  MoveL 604 to (474.95, 542.05, 8) mm, rotated rx 180 ry 0 rz 160 deg; joints [12.107, 76.051, -6.666, -146.162, 72.648, 168.694]
  Set speed (17.5 mm/s)
  Call Extruder(1520.11430)
  MoveL 605 to (474.5, 541.77, 8) mm, rotated rx 180 ry 0 rz 160 deg; joints [12.084, 75.99, -6.51, -146.202, 72.722, 168.756]
  Set speed (17.5 mm/s)
  Call Extruder(1525.02025)
  MoveL 606 to (473.22, 540.96, 8) mm, rotated rx 180 ry 0 rz 160 deg; joints [12.014, 75.813, -6.063, -146.32, 72.934, 168.934]
  Set speed (17.5 mm/s)
  Call Extruder(1527.82496)
  MoveL 607 to (472.5, 540.48, 8) mm, rotated rx 180 ry 0 rz 160 deg; joints [11.972, 75.714, -5.811, -146.39, 73.053, 169.035]
  Set speed (17.4 mm/s)
  Call Extruder(1533.06308)
  MoveL 608 to (471.18, 539.55, 8) mm, rotated rx -180 ry 0 rz 160 deg; joints [11.887, 75.532, -5.348, -146.524, 73.271, 169.223]
  Set speed (17.4 mm/s)
  Call Extruder(1536.34508)
  MoveL 609 to (470.36, 538.94, 8) mm, rotated rx 180 ry 0 rz 160 deg; joints [11.83, 75.421, -5.064, -146.611, 73.405, 169.339]
  Set speed (17.4 mm/s)
  Call Extruder(1538.57380)
  MoveL 610 to (469.82, 538.52, 8) mm, rotated rx 180 ry 0 rz 160 deg; joints [11.79, 75.346, -4.872, -146.671, 73.495, 169.418]
  Set speed (17.5 mm/s)
  Call Extruder(1541.82142)
  MoveL 611 to (469.03, 537.89, 8) mm, rotated rx -180 ry 0 rz 160 deg; joints [11.729, 75.239, -4.597, -146.761, 73.625, 169.532]
  Set speed (17.5 mm/s)
  Call Extruder(1547.90773)
  MoveL 612 to (467.59, 536.68, 8) mm, rotated rx 180 ry 0 rz 160 deg; joints [11.608, 75.042, -4.09, -146.934, 73.863, 169.743]
  Set speed (17.5 mm/s)
  Call Extruder(1552.51952)
  MoveL 613 to (466.54, 535.71, 8) mm, rotated rx 180 ry 0 rz 160 deg; joints [11.509, 74.899, -3.717, -147.071, 74.037, 169.901]
  Set speed (17.4 mm/s)
  Call Extruder(1558.05894)
  MoveL 614 to (465.31, 534.52, 8) mm, rotated rx -180 ry 0 rz 160 deg; joints [11.384, 74.731, -3.281, -147.241, 74.241, 170.087]
  Set speed (17.5 mm/s)
  Call Extruder(1561.63478)
  MoveL 615 to (464.54, 533.73, 8) mm, rotated rx 180 ry 0 rz 160 deg; joints [11.299, 74.625, -3.007, -147.353, 74.369, 170.206]
  Call Extruder(1565.31804)
  MoveL 616 to (463.76, 532.89, 8) mm, rotated rx -180 ry 0 rz 160 deg; joints [11.208, 74.519, -2.73, -147.472, 74.497, 170.326]
  Set speed (17.5 mm/s)
  Call Extruder(1568.71161)
  MoveL 617 to (463.07, 532.11, 8) mm, rotated rx 180 ry 0 rz 160 deg; joints [11.122, 74.424, -2.479, -147.583, 74.614, 170.436]
  Call Extruder(0.00000)
  Set speed (17.4 mm/s)
  Call Extruder(3.82302)
  MoveL 618 to (462.3, 531.2, 8) mm, rotated rx 180 ry 0 rz 160 deg; joints [11.021, 74.319, -2.204, -147.711, 74.741, 170.558]
  Set speed (17.5 mm/s)
  Call Extruder(8.69578)
  MoveL 619 to (461.36, 530.03, 8) mm, rotated rx 180 ry 0 rz 160 deg; joints [10.888, 74.19, -1.863, -147.878, 74.898, 170.71]
  Set speed (17.5 mm/s)
  Call Extruder(11.81632)
  MoveL 620 to (460.77, 529.26, 8) mm, rotated rx 180 ry 0 rz 160 deg; joints [10.799, 74.109, -1.65, -147.988, 74.996, 170.807]
  Set speed (17.5 mm/s)
  Call Extruder(16.00361)
  MoveL 621 to (460.01, 528.21, 8) mm, rotated rx 180 ry 0 rz 160 deg; joints [10.677, 74.004, -1.372, -148.137, 75.124, 170.934]
  Set speed (17.5 mm/s)
  Call Extruder(19.39363)
  MoveL 622 to (459.42, 527.35, 8) mm, rotated rx 180 ry 0 rz 160 deg; joints [10.575, 73.922, -1.153, -148.26, 75.224, 171.035]
  Set speed (17.5 mm/s)
  Call Extruder(23.27967)
  MoveL 623 to (458.76, 526.34, 8) mm, rotated rx 180 ry 0 rz 160 deg; joints [10.456, 73.83, -0.91, -148.403, 75.335, 171.148]
  Set speed (17.5 mm/s)
  Call Extruder(28.16959)
  MoveL 624 to (457.96, 525.05, 8) mm, rotated rx 180 ry 0 rz 160 deg; joints [10.3, 73.72, -0.614, -148.587, 75.469, 171.288]
  Call Extruder(32.04491)
  MoveL 625 to (457.36, 524.02, 8) mm, rotated rx -180 ry 0 rz 160 deg; joints [10.174, 73.635, -0.388, -148.735, 75.571, 171.397]
  Set speed (17.5 mm/s)
  Call Extruder(35.64970)
  MoveL 626 to (456.83, 523.04, 8) mm, rotated rx 180 ry 0 rz 160 deg; joints [10.053, 73.559, -0.184, -148.875, 75.662, 171.495]
  Call Extruder(38.75076)
  MoveL 627 to (456.38, 522.19, 8) mm, rotated rx -180 ry 0 rz 160 deg; joints [9.948, 73.497, -0.015, -148.997, 75.738, 171.579]
  Set speed (17.4 mm/s)
  Call Extruder(42.04623)
  MoveL 628 to (455.93, 521.28, 8) mm, rotated rx 180 ry 0 rz 160 deg; joints [9.833, 73.432, 0.159, -149.128, 75.815, 171.665]
  Set speed (17.4 mm/s)
  Call Extruder(45.26649)
  MoveL 629 to (455.51, 520.38, 8) mm, rotated rx 180 ry 0 rz 160 deg; joints [9.719, 73.371, 0.323, -149.258, 75.887, 171.748]
  Set speed (17.4 mm/s)
  Call Extruder(48.51642)
  MoveL 630 to (455.1, 519.46, 8) mm, rotated rx 180 ry 0 rz 160 deg; joints [9.603, 73.312, 0.484, -149.389, 75.958, 171.831]
  Set speed (17.4 mm/s)
  Call Extruder(52.84820)
  MoveL 631 to (454.58, 518.22, 8) mm, rotated rx -180 ry 0 rz 160 deg; joints [9.444, 73.236, 0.689, -149.568, 76.047, 171.937]
  Set speed (17.5 mm/s)
  Call Extruder(59.01689)
  MoveL 632 to (453.9, 516.44, 8) mm, rotated rx -180 ry 0 rz 160 deg; joints [9.213, 73.135, 0.964, -149.825, 76.164, 172.084]
  Set speed (17.5 mm/s)
  Call Extruder(61.45313)
  MoveL 633 to (453.66, 515.72, 8) mm, rotated rx -180 ry 0 rz 160 deg; joints [9.119, 73.098, 1.064, -149.928, 76.207, 172.14]
  Set speed (17.4 mm/s)
  Call Extruder(67.12764)
  MoveL 634 to (453.12, 514.05, 8) mm, rotated rx 180 ry 0 rz 160 deg; joints [8.899, 73.015, 1.29, -150.17, 76.301, 172.267]
  Set speed (17.4 mm/s)
  Call Extruder(71.17621)
  MoveL 635 to (452.78, 512.85, 8) mm, rotated rx -180 ry 0 rz 160 deg; joints [8.739, 72.961, 1.438, -150.345, 76.361, 172.353]
  Set speed (17.4 mm/s)
  Call Extruder(74.29378)
  MoveL 636 to (452.53, 511.92, 8) mm, rotated rx -180 ry 0 rz 160 deg; joints [8.615, 72.921, 1.548, -150.48, 76.405, 172.419]
  Set speed (17.4 mm/s)
  Call Extruder(77.03216)
  MoveL 637 to (452.34, 511.1, 8) mm, rotated rx 180 ry 0 rz 160 deg; joints [8.504, 72.888, 1.637, -150.6, 76.44, 172.474]
  Set speed (17.4 mm/s)
  Call Extruder(81.46566)
  MoveL 638 to (452.05, 509.76, 8) mm, rotated rx 180 ry 0 rz 160 deg; joints [8.324, 72.838, 1.775, -150.794, 76.493, 172.561]
  Set speed (17.4 mm/s)
  Call Extruder(87.40179)
  MoveL 639 to (451.72, 507.96, 8) mm, rotated rx 180 ry 0 rz 160 deg; joints [8.078, 72.778, 1.94, -151.057, 76.553, 172.672]
  Set speed (17.5 mm/s)
  Call Extruder(91.56460)
  MoveL 640 to (451.53, 506.68, 8) mm, rotated rx -180 ry 0 rz 160 deg; joints [7.903, 72.741, 2.043, -151.243, 76.589, 172.746]
  Set speed (17.5 mm/s)
  Call Extruder(93.86761)
  MoveL 641 to (451.43, 505.98, 8) mm, rotated rx 180 ry 0 rz 160 deg; joints [7.806, 72.721, 2.097, -151.346, 76.606, 172.786]
  Set speed (17.4 mm/s)
  Call Extruder(100.33911)
  MoveL 642 to (451.23, 503.99, 8) mm, rotated rx -180 ry 0 rz 160 deg; joints [7.53, 72.673, 2.229, -151.636, 76.646, 172.892]
  Set speed (17.5 mm/s)
  Call Extruder(105.92398)
  MoveL 643 to (451.12, 502.26, 8) mm, rotated rx 180 ry 0 rz 160 deg; joints [7.29, 72.64, 2.322, -151.888, 76.669, 172.978]
  Set speed (17.5 mm/s)
  Call Extruder(108.19606)
  MoveL 644 to (451.09, 501.56, 8) mm, rotated rx 180 ry 0 rz 160 deg; joints [7.191, 72.628, 2.354, -151.991, 76.675, 173.011]
  Set speed (17.5 mm/s)
  Call Extruder(113.19534)
  MoveL 645 to (451.06, 500.01, 8) mm, rotated rx -180 ry 0 rz 160 deg; joints [6.974, 72.606, 2.416, -152.218, 76.683, 173.081]
  Set speed (17.4 mm/s)
  Call Extruder(119.10860)
  MoveL 646 to (451.1, 498.18, 8) mm, rotated rx -180 ry 0 rz 160 deg; joints [6.715, 72.587, 2.467, -152.485, 76.681, 173.157]
  Set speed (17.4 mm/s)
  Call Extruder(124.85256)
  MoveL 647 to (451.2, 496.41, 8) mm, rotated rx 180 ry 0 rz 160 deg; joints [6.463, 72.577, 2.497, -152.744, 76.668, 173.225]
  Set speed (17.5 mm/s)
  Call Extruder(129.53981)
  MoveL 648 to (451.32, 494.97, 8) mm, rotated rx 180 ry 0 rz 160 deg; joints [6.257, 72.573, 2.506, -152.955, 76.649, 173.277]
  Set speed (17.5 mm/s)
  Call Extruder(136.75028)
  MoveL 649 to (451.6, 492.76, 8) mm, rotated rx 180 ry 0 rz 160 deg; joints [5.94, 72.578, 2.494, -153.278, 76.606, 173.348]
  Set speed (17.4 mm/s)
  Call Extruder(142.41552)
  MoveL 650 to (451.89, 491.03, 8) mm, rotated rx -180 ry 0 rz 160 deg; joints [5.692, 72.589, 2.462, -153.529, 76.559, 173.398]
  Set speed (17.4 mm/s)
  Call Extruder(148.15055)
  MoveL 651 to (452.25, 489.29, 8) mm, rotated rx 180 ry 0 rz 160 deg; joints [5.442, 72.608, 2.409, -153.781, 76.5, 173.442]
  Set speed (17.4 mm/s)
  Call Extruder(153.97860)
  MoveL 652 to (452.68, 487.54, 8) mm, rotated rx -180 ry 0 rz 160 deg; joints [5.189, 72.635, 2.336, -154.035, 76.429, 173.481]
  Set speed (17.5 mm/s)
  Call Extruder(159.80113)
  MoveL 653 to (453.17, 485.81, 8) mm, rotated rx 180 ry 0 rz 160 deg; joints [4.937, 72.669, 2.242, -154.285, 76.346, 173.515]
  Set speed (17.5 mm/s)
  Call Extruder(165.63454)
  MoveL 654 to (453.72, 484.09, 8) mm, rotated rx -180 ry 0 rz 160 deg; joints [4.688, 72.711, 2.127, -154.532, 76.252, 173.542]
  Call Extruder(171.46465)
  MoveL 655 to (454.34, 482.4, 8) mm, rotated rx -180 ry 0 rz 160 deg; joints [4.442, 72.76, 1.992, -154.775, 76.146, 173.564]
  Set speed (17.4 mm/s)
  Call Extruder(176.47279)
  MoveL 656 to (454.91, 480.96, 8) mm, rotated rx 180 ry 0 rz 160 deg; joints [4.233, 72.807, 1.86, -154.98, 76.047, 173.579]
  Call Extruder(183.18953)
  MoveL 657 to (455.77, 479.07, 8) mm, rotated rx 180 ry 0 rz 160 deg; joints [3.958, 72.881, 1.657, -155.249, 75.9, 173.592]
  Call Extruder(188.92581)
  MoveL 658 to (456.56, 477.48, 8) mm, rotated rx 180 ry 0 rz 160 deg; joints [3.727, 72.952, 1.464, -155.473, 75.762, 173.597]
  Set speed (17.5 mm/s)
  Call Extruder(192.53165)
  MoveL 659 to (457.08, 476.5, 8) mm, rotated rx 180 ry 0 rz 160 deg; joints [3.584, 73, 1.332, -155.61, 75.67, 173.597]
  Call Extruder(194.75891)
  MoveL 660 to (457.42, 475.89, 8) mm, rotated rx -180 ry 0 rz 160 deg; joints [3.497, 73.031, 1.247, -155.694, 75.611, 173.596]
  Set speed (17.5 mm/s)
  Call Extruder(200.05688)
  MoveL 661 to (458.24, 474.48, 8) mm, rotated rx -180 ry 0 rz 160 deg; joints [3.291, 73.108, 1.036, -155.891, 75.466, 173.592]
  Set speed (17.5 mm/s)
  Call Extruder(206.40402)
  MoveL 662 to (459.3, 472.82, 8) mm, rotated rx -180 ry 0 rz 160 deg; joints [3.051, 73.21, 0.76, -156.119, 75.28, 173.581]
  Set speed (17.5 mm/s)
  Call Extruder(213.20115)
  MoveL 663 to (460.51, 471.1, 8) mm, rotated rx 180 ry 0 rz 160 deg; joints [2.802, 73.328, 0.439, -156.353, 75.067, 173.562]
  Set speed (17.4 mm/s)
  Call Extruder(218.13202)
  MoveL 664 to (461.43, 469.89, 8) mm, rotated rx -180 ry 0 rz 160 deg; joints [2.627, 73.42, 0.19, -156.517, 74.903, 173.544]
  Set speed (17.4 mm/s)
  Call Extruder(223.87123)
  MoveL 665 to (462.55, 468.51, 8) mm, rotated rx 180 ry 0 rz 160 deg; joints [2.428, 73.533, -0.114, -156.701, 74.705, 173.519]
  Set speed (17.5 mm/s)
  Call Extruder(229.75874)
  MoveL 666 to (463.74, 467.13, 8) mm, rotated rx -180 ry 0 rz 160 deg; joints [2.231, 73.657, -0.445, -156.881, 74.492, 173.488]
  Set speed (17.4 mm/s)
  Call Extruder(235.61813)
  MoveL 667 to (464.98, 465.81, 8) mm, rotated rx 180 ry 0 rz 160 deg; joints [2.042, 73.787, -0.793, -157.052, 74.27, 173.452]
  Set speed (17.4 mm/s)
  Call Extruder(241.35830)
  MoveL 668 to (466.25, 464.57, 8) mm, rotated rx 180 ry 0 rz 160 deg; joints [1.865, 73.921, -1.15, -157.211, 74.044, 173.412]
  Set speed (17.5 mm/s)
  Call Extruder(243.43277)
  MoveL 669 to (466.72, 464.13, 8) mm, rotated rx 180 ry 0 rz 160 deg; joints [1.802, 73.971, -1.284, -157.267, 73.96, 173.396]
  Set speed (17.4 mm/s)
  Call Extruder(247.19209)
  MoveL 670 to (467.58, 463.35, 8) mm, rotated rx 180 ry 0 rz 160 deg; joints [1.691, 74.064, -1.53, -157.364, 73.806, 173.367]
  Set speed (17.4 mm/s)
  Call Extruder(253.10581)
  MoveL 671 to (468.96, 462.16, 8) mm, rotated rx 180 ry 0 rz 160 deg; joints [1.523, 74.215, -1.931, -157.51, 73.557, 173.316]
  Call Extruder(259.12323)
  MoveL 672 to (470.42, 461.01, 8) mm, rotated rx 180 ry 0 rz 160 deg; joints [1.361, 74.377, -2.356, -157.649, 73.294, 173.259]
  Set speed (17.4 mm/s)
  Call Extruder(264.11346)
  MoveL 673 to (471.67, 460.1, 8) mm, rotated rx 180 ry 0 rz 160 deg; joints [1.233, 74.516, -2.721, -157.755, 73.07, 173.208]
  Set speed (17.4 mm/s)
  Call Extruder(270.55259)
  MoveL 674 to (473.31, 458.98, 8) mm, rotated rx -180 ry 0 rz 160 deg; joints [1.077, 74.703, -3.208, -157.883, 72.773, 173.137]
  Set speed (17.4 mm/s)
  Call Extruder(276.42854)
  MoveL 675 to (474.85, 458.02, 8) mm, rotated rx 180 ry 0 rz 160 deg; joints [0.942, 74.88, -3.669, -157.989, 72.494, 173.067]
  Set speed (17.4 mm/s)
  Call Extruder(282.26197)
  MoveL 676 to (476.42, 457.12, 8) mm, rotated rx -180 ry 0 rz 160 deg; joints [0.818, 75.062, -4.14, -158.084, 72.211, 172.992]
  Set speed (17.4 mm/s)
  Call Extruder(288.04120)
  MoveL 677 to (478, 456.29, 8) mm, rotated rx 180 ry 0 rz 160 deg; joints [0.703, 75.248, -4.62, -158.168, 71.924, 172.914]
  Set speed (17.4 mm/s)
  Call Extruder(293.86773)
  MoveL 678 to (479.62, 455.51, 8) mm, rotated rx 180 ry 0 rz 160 deg; joints [0.597, 75.442, -5.118, -158.242, 71.629, 172.831]
  Call Extruder(299.75358)
  MoveL 679 to (481.29, 454.78, 8) mm, rotated rx 180 ry 0 rz 160 deg; joints [0.498, 75.644, -5.633, -158.307, 71.325, 172.741]
  Set speed (17.4 mm/s)
  Call Extruder(305.48396)
  MoveL 680 to (482.94, 454.14, 8) mm, rotated rx -180 ry 0 rz 160 deg; joints [0.41, 75.846, -6.145, -158.36, 71.025, 172.649]
  Set speed (17.4 mm/s)
  Call Extruder(311.35103)
  MoveL 681 to (484.65, 453.54, 8) mm, rotated rx 180 ry 0 rz 160 deg; joints [0.329, 76.058, -6.682, -158.403, 70.713, 172.551]
  Call Extruder(317.21255)
  MoveL 682 to (486.37, 453, 8) mm, rotated rx 180 ry 0 rz 160 deg; joints [0.258, 76.274, -7.228, -158.436, 70.398, 172.447]
  Set speed (17.4 mm/s)
  Call Extruder(322.81686)
  MoveL 683 to (488.05, 452.55, 8) mm, rotated rx 180 ry 0 rz 160 deg; joints [0.197, 76.487, -7.761, -158.457, 70.092, 172.344]
  Set speed (17.4 mm/s)
  Call Extruder(328.90646)
  MoveL 684 to (489.88, 452.12, 8) mm, rotated rx 180 ry 0 rz 160 deg; joints [0.141, 76.723, -8.35, -158.469, 69.756, 172.226]
  Set speed (17.5 mm/s)
  Call Extruder(332.37006)
  MoveL 685 to (490.93, 451.91, 8) mm, rotated rx 180 ry 0 rz 160 deg; joints [0.113, 76.86, -8.69, -158.471, 69.563, 172.157]
  Set speed (17.5 mm/s)
  Call Extruder(334.62537)
  MoveL 686 to (491.62, 451.79, 8) mm, rotated rx -180 ry 0 rz 160 deg; joints [0.097, 76.95, -8.913, -158.47, 69.437, 172.111]
  Set speed (17.4 mm/s)
  Call Extruder(340.25590)
  MoveL 687 to (493.33, 451.52, 8) mm, rotated rx -180 ry 0 rz 160 deg; joints [0.062, 77.177, -9.474, -158.461, 69.121, 171.993]
  Set speed (17.4 mm/s)
  Call Extruder(346.16641)
  MoveL 688 to (495.15, 451.3, 8) mm, rotated rx 180 ry 0 rz 160 deg; joints [0.034, 77.419, -10.072, -158.44, 68.787, 171.864]
  Set speed (17.5 mm/s)
  Call Extruder(352.11718)
  MoveL 689 to (496.99, 451.15, 8) mm, rotated rx -180 ry 0 rz 160 deg; joints [0.014, 77.668, -10.682, -158.409, 68.448, 171.729]
  Set speed (17.5 mm/s)
  Call Extruder(358.01649)
  MoveL 690 to (498.81, 451.08, 8) mm, rotated rx -180 ry 0 rz 160 deg; joints [0.004, 77.919, -11.293, -158.366, 68.111, 171.589]
  Set speed (17.4 mm/s)
  Call Extruder(363.77984)
  MoveL 691 to (500.59, 451.07, 8) mm, rotated rx 180 ry 0 rz 160 deg; joints [0.003, 78.167, -11.896, -158.315, 67.782, 171.449]
  Set speed (17.5 mm/s)
  Call Extruder(369.76327)
  MoveL 692 to (502.44, 451.12, 8) mm, rotated rx 180 ry 0 rz 160 deg; joints [0.01, 78.428, -12.527, -158.251, 67.439, 171.298]
  Set speed (17.5 mm/s)
  Call Extruder(375.43569)
  MoveL 693 to (504.19, 451.24, 8) mm, rotated rx -180 ry 0 rz 160 deg; joints [0.026, 78.678, -13.13, -158.18, 67.114, 171.15]
  Set speed (17.4 mm/s)
  Call Extruder(381.32270)
  MoveL 694 to (506, 451.43, 8) mm, rotated rx -180 ry 0 rz 160 deg; joints [0.049, 78.94, -13.759, -158.096, 66.778, 170.991]
  Set speed (17.5 mm/s)
  Call Extruder(385.86187)
  MoveL 695 to (507.39, 451.63, 8) mm, rotated rx 180 ry 0 rz 160 deg; joints [0.073, 79.145, -14.246, -158.024, 66.518, 170.866]
  Set speed (17.5 mm/s)
  Call Extruder(392.76070)
  MoveL 696 to (509.5, 451.99, 8) mm, rotated rx 180 ry 0 rz 160 deg; joints [0.119, 79.458, -14.991, -157.905, 66.126, 170.669]
  Set speed (17.4 mm/s)
  Call Extruder(398.73898)
  MoveL 697 to (511.3, 452.39, 8) mm, rotated rx 180 ry 0 rz 160 deg; joints [0.167, 79.73, -15.637, -157.789, 65.788, 170.494]
  Set speed (17.4 mm/s)
  Call Extruder(404.54907)
  MoveL 698 to (513.04, 452.84, 8) mm, rotated rx 180 ry 0 rz 160 deg; joints [0.222, 79.997, -16.265, -157.668, 65.462, 170.319]
  Call Extruder(410.41827)
  MoveL 699 to (514.78, 453.35, 8) mm, rotated rx -180 ry 0 rz 160 deg; joints [0.285, 80.268, -16.901, -157.536, 65.135, 170.137]
  Set speed (17.5 mm/s)
  Call Extruder(416.23130)
  MoveL 700 to (516.49, 453.92, 8) mm, rotated rx 180 ry 0 rz 160 deg; joints [0.354, 80.536, -17.53, -157.396, 64.814, 169.953]
  Call Extruder(422.02291)
  MoveL 701 to (518.16, 454.56, 8) mm, rotated rx -180 ry 0 rz 160 deg; joints [0.431, 80.804, -18.155, -157.247, 64.499, 169.765]
  Set speed (17.4 mm/s)
  Call Extruder(427.93868)
  MoveL 702 to (519.84, 455.27, 8) mm, rotated rx -180 ry 0 rz 160 deg; joints [0.516, 81.078, -18.791, -157.087, 64.18, 169.569]
  Set speed (17.5 mm/s)
  Call Extruder(430.83975)
  MoveL 703 to (520.66, 455.64, 8) mm, rotated rx -180 ry 0 rz 160 deg; joints [0.561, 81.213, -19.102, -157.005, 64.026, 169.471]
  Call Extruder(433.75248)
  MoveL 704 to (521.47, 456.03, 8) mm, rotated rx 180 ry 0 rz 160 deg; joints [0.607, 81.347, -19.413, -156.92, 63.872, 169.372]
  Set speed (17.4 mm/s)
  Call Extruder(439.48747)
  MoveL 705 to (523.06, 456.83, 8) mm, rotated rx 180 ry 0 rz 160 deg; joints [0.702, 81.612, -20.023, -156.748, 63.572, 169.174]
  Call Extruder(445.40417)
  MoveL 706 to (524.65, 457.73, 8) mm, rotated rx 180 ry 0 rz 160 deg; joints [0.808, 81.883, -20.646, -156.562, 63.269, 168.966]
  Set speed (17.4 mm/s)
  Call Extruder(451.15607)
  MoveL 707 to (526.17, 458.65, 8) mm, rotated rx -180 ry 0 rz 160 deg; joints [0.917, 82.145, -21.247, -156.374, 62.98, 168.76]
  Set speed (17.4 mm/s)
  Call Extruder(456.43020)
  MoveL 708 to (527.53, 459.54, 8) mm, rotated rx 180 ry 0 rz 160 deg; joints [1.021, 82.385, -21.793, -156.196, 62.719, 168.569]
  Set speed (17.4 mm/s)
  Call Extruder(462.80027)
  MoveL 709 to (529.14, 460.68, 8) mm, rotated rx -180 ry 0 rz 160 deg; joints [1.154, 82.671, -22.444, -155.972, 62.412, 168.335]
  Call Extruder(468.64160)
  MoveL 710 to (530.57, 461.79, 8) mm, rotated rx -180 ry 0 rz 160 deg; joints [1.283, 82.93, -23.031, -155.76, 62.139, 168.117]
  Call Extruder(474.55020)
  MoveL 711 to (531.97, 462.95, 8) mm, rotated rx -180 ry 0 rz 160 deg; joints [1.418, 83.189, -23.617, -155.539, 61.87, 167.895]
  Set speed (17.5 mm/s)
  Call Extruder(479.16625)
  MoveL 712 to (533.04, 463.9, 8) mm, rotated rx -180 ry 0 rz 160 deg; joints [1.528, 83.389, -24.067, -155.361, 61.665, 167.719]
  Set speed (17.5 mm/s)
  Call Extruder(480.82756)
  MoveL 713 to (533.42, 464.25, 8) mm, rotated rx -180 ry 0 rz 160 deg; joints [1.568, 83.46, -24.227, -155.296, 61.593, 167.655]
  Set speed (17.4 mm/s)
  Call Extruder(486.22558)
  MoveL 714 to (534.62, 465.41, 8) mm, rotated rx -180 ry 0 rz 160 deg; joints [1.701, 83.689, -24.743, -155.083, 61.362, 167.448]
  Set speed (17.4 mm/s)
  Call Extruder(489.36043)
  MoveL 715 to (535.29, 466.11, 8) mm, rotated rx -180 ry 0 rz 160 deg; joints [1.781, 83.819, -25.034, -154.957, 61.233, 167.328]
  Set speed (17.5 mm/s)
  Call Extruder(493.94205)
  MoveL 716 to (536.27, 467.14, 8) mm, rotated rx 180 ry 0 rz 160 deg; joints [1.899, 84.01, -25.46, -154.771, 61.046, 167.15]
  Set speed (17.5 mm/s)
  Call Extruder(500.40882)
  MoveL 717 to (537.58, 468.65, 8) mm, rotated rx 180 ry 0 rz 160 deg; joints [2.071, 84.271, -26.043, -154.501, 60.794, 166.899]
  Set speed (17.5 mm/s)
  Call Extruder(502.32242)
  MoveL 718 to (537.95, 469.11, 8) mm, rotated rx -180 ry 0 rz 160 deg; joints [2.123, 84.346, -26.212, -154.421, 60.722, 166.825]
  Set speed (17.4 mm/s)
  Call Extruder(505.53291)
  MoveL 719 to (538.57, 469.89, 8) mm, rotated rx -180 ry 0 rz 160 deg; joints [2.212, 84.471, -26.49, -154.285, 60.604, 166.7]
  Set speed (17.5 mm/s)
  Call Extruder(509.69795)
  MoveL 720 to (539.35, 470.91, 8) mm, rotated rx -180 ry 0 rz 160 deg; joints [2.328, 84.633, -26.848, -154.106, 60.453, 166.538]
  Set speed (17.5 mm/s)
  Call Extruder(512.03969)
  MoveL 721 to (539.78, 471.5, 8) mm, rotated rx 180 ry 0 rz 160 deg; joints [2.395, 84.721, -27.043, -154.005, 60.372, 166.447]
  Set speed (17.4 mm/s)
  Call Extruder(517.54038)
  MoveL 722 to (540.75, 472.89, 8) mm, rotated rx 180 ry 0 rz 160 deg; joints [2.553, 84.926, -27.498, -153.766, 60.186, 166.233]
  Set speed (17.5 mm/s)
  Call Extruder(523.34543)
  MoveL 723 to (541.71, 474.41, 8) mm, rotated rx 180 ry 0 rz 160 deg; joints [2.725, 85.132, -27.955, -153.509, 60.002, 166.008]
  Set speed (17.5 mm/s)
  Call Extruder(526.58606)
  MoveL 724 to (542.23, 475.27, 8) mm, rotated rx 180 ry 0 rz 160 deg; joints [2.822, 85.245, -28.205, -153.365, 59.904, 165.884]
  Call Extruder(532.05474)
  MoveL 725 to (543.05, 476.74, 8) mm, rotated rx 180 ry 0 rz 160 deg; joints [2.988, 85.429, -28.61, -153.121, 59.747, 165.674]
  Set speed (17.5 mm/s)
  Call Extruder(536.96359)
  MoveL 726 to (543.76, 478.09, 8) mm, rotated rx -180 ry 0 rz 160 deg; joints [3.14, 85.589, -28.961, -152.9, 59.614, 165.488]
  Set speed (17.5 mm/s)
  Call Extruder(541.13842)
  MoveL 727 to (544.32, 479.25, 8) mm, rotated rx -180 ry 0 rz 160 deg; joints [3.271, 85.719, -29.247, -152.711, 59.508, 165.331]
  Set speed (17.5 mm/s)
  Call Extruder(544.43131)
  MoveL 728 to (544.75, 480.18, 8) mm, rotated rx 180 ry 0 rz 160 deg; joints [3.375, 85.819, -29.465, -152.561, 59.429, 165.208]
  Set speed (17.5 mm/s)
  Call Extruder(549.20774)
  MoveL 729 to (545.32, 481.54, 8) mm, rotated rx 180 ry 0 rz 160 deg; joints [3.528, 85.957, -29.769, -152.344, 59.322, 165.031]
  Set speed (17.4 mm/s)
  Call Extruder(554.07983)
  MoveL 730 to (545.87, 482.94, 8) mm, rotated rx 180 ry 0 rz 160 deg; joints [3.686, 86.09, -30.061, -152.123, 59.223, 164.855]
  Set speed (17.4 mm/s)
  Call Extruder(556.54437)
  MoveL 731 to (546.13, 483.66, 8) mm, rotated rx -180 ry 0 rz 160 deg; joints [3.766, 86.157, -30.206, -152.011, 59.175, 164.766]
  Set speed (17.4 mm/s)
  Call Extruder(560.55299)
  MoveL 732 to (546.52, 484.83, 8) mm, rotated rx 180 ry 0 rz 160 deg; joints [3.899, 86.257, -30.426, -151.829, 59.104, 164.624]
  Set speed (17.4 mm/s)
  Call Extruder(563.65651)
  MoveL 733 to (546.82, 485.75, 8) mm, rotated rx 180 ry 0 rz 160 deg; joints [4.001, 86.334, -30.593, -151.688, 59.052, 164.515]
  Set speed (17.4 mm/s)
  Call Extruder(570.27664)
  MoveL 734 to (547.37, 487.71, 8) mm, rotated rx -180 ry 0 rz 160 deg; joints [4.223, 86.484, -30.92, -151.388, 58.956, 164.288]
  Set speed (17.4 mm/s)
  Call Extruder(573.49816)
  MoveL 735 to (547.61, 488.68, 8) mm, rotated rx 180 ry 0 rz 160 deg; joints [4.332, 86.551, -31.067, -151.243, 58.915, 164.18]
  Call Extruder(576.77004)
  MoveL 736 to (547.83, 489.67, 8) mm, rotated rx 180 ry 0 rz 160 deg; joints [4.443, 86.616, -31.208, -151.096, 58.879, 164.073]
  Set speed (17.5 mm/s)
  Call Extruder(580.90913)
  MoveL 737 to (548.08, 490.92, 8) mm, rotated rx 180 ry 0 rz 160 deg; joints [4.584, 86.693, -31.375, -150.91, 58.839, 163.94]
  Call Extruder(583.21130)
  MoveL 738 to (548.21, 491.62, 8) mm, rotated rx -180 ry 0 rz 160 deg; joints [4.663, 86.734, -31.464, -150.808, 58.819, 163.866]
  Set speed (17.4 mm/s)
  Call Extruder(589.67407)
  MoveL 739 to (548.51, 493.6, 8) mm, rotated rx -180 ry 0 rz 160 deg; joints [4.886, 86.837, -31.688, -150.522, 58.776, 163.668]
  Set speed (17.5 mm/s)
  Call Extruder(596.24528)
  MoveL 740 to (548.74, 495.62, 8) mm, rotated rx 180 ry 0 rz 160 deg; joints [5.114, 86.926, -31.882, -150.234, 58.75, 163.474]
  Set speed (17.5 mm/s)
  Call Extruder(602.63347)
  MoveL 741 to (548.88, 497.59, 8) mm, rotated rx 180 ry 0 rz 160 deg; joints [5.338, 86.997, -32.035, -149.958, 58.742, 163.296]
  Set speed (17.5 mm/s)
  Call Extruder(609.09670)
  MoveL 742 to (548.93, 499.59, 8) mm, rotated rx -180 ry 0 rz 160 deg; joints [5.565, 87.052, -32.155, -149.684, 58.752, 163.126]
  Set speed (17.4 mm/s)
  Call Extruder(615.66386)
  MoveL 743 to (548.91, 501.62, 8) mm, rotated rx -180 ry 0 rz 160 deg; joints [5.796, 87.091, -32.24, -149.411, 58.78, 162.965]
  Set speed (17.5 mm/s)
  Call Extruder(619.76956)
  MoveL 744 to (548.85, 502.89, 8) mm, rotated rx 180 ry 0 rz 160 deg; joints [5.942, 87.107, -32.274, -149.244, 58.807, 162.87]
  Set speed (17.4 mm/s)
  Call Extruder(622.04137)
  MoveL 745 to (548.8, 503.59, 8) mm, rotated rx -180 ry 0 rz 160 deg; joints [6.022, 87.113, -32.287, -149.152, 58.824, 162.819]
  Set speed (17.4 mm/s)
  Call Extruder(627.80930)
  MoveL 746 to (548.64, 505.36, 8) mm, rotated rx 180 ry 0 rz 160 deg; joints [6.226, 87.12, -32.303, -148.922, 58.877, 162.697]
  Set speed (17.4 mm/s)
  Call Extruder(635.09938)
  MoveL 747 to (548.34, 507.59, 8) mm, rotated rx -180 ry 0 rz 160 deg; joints [6.483, 87.108, -32.277, -148.639, 58.966, 162.557]
  Set speed (17.5 mm/s)
  Call Extruder(641.47666)
  MoveL 748 to (548, 509.53, 8) mm, rotated rx -180 ry 0 rz 160 deg; joints [6.708, 87.082, -32.219, -148.398, 59.06, 162.447]
  Set speed (17.5 mm/s)
  Call Extruder(648.66448)
  MoveL 749 to (547.52, 511.71, 8) mm, rotated rx 180 ry 0 rz 160 deg; joints [6.962, 87.033, -32.113, -148.135, 59.186, 162.338]
  Set speed (17.5 mm/s)
  Call Extruder(654.43022)
  MoveL 750 to (547.06, 513.43, 8) mm, rotated rx 180 ry 0 rz 160 deg; joints [7.164, 86.978, -31.995, -147.931, 59.301, 162.262]
  Call Extruder(656.37140)
  MoveL 751 to (546.89, 514.01, 8) mm, rotated rx -180 ry 0 rz 160 deg; joints [7.232, 86.957, -31.948, -147.863, 59.343, 162.239]
  Set speed (17.5 mm/s)
  Call Extruder(660.77672)
  MoveL 752 to (546.48, 515.31, 8) mm, rotated rx 180 ry 0 rz 160 deg; joints [7.386, 86.904, -31.833, -147.713, 59.443, 162.191]
  Set speed (17.4 mm/s)
  Call Extruder(664.14135)
  MoveL 753 to (546.14, 516.29, 8) mm, rotated rx 180 ry 0 rz 160 deg; joints [7.503, 86.857, -31.732, -147.601, 59.525, 162.159]
  Set speed (17.4 mm/s)
  Call Extruder(667.39027)
  MoveL 754 to (545.8, 517.23, 8) mm, rotated rx -180 ry 0 rz 160 deg; joints [7.615, 86.809, -31.628, -147.495, 59.607, 162.132]
  Set speed (17.5 mm/s)
  Call Extruder(673.00051)
  MoveL 755 to (545.16, 518.85, 8) mm, rotated rx 180 ry 0 rz 160 deg; joints [7.808, 86.718, -31.43, -147.315, 59.756, 162.091]
  Set speed (17.4 mm/s)
  Call Extruder(677.09149)
  MoveL 756 to (544.65, 520.01, 8) mm, rotated rx -180 ry 0 rz 160 deg; joints [7.948, 86.642, -31.265, -147.189, 59.874, 162.069]
  Set speed (17.4 mm/s)
  Call Extruder(680.67724)
  MoveL 757 to (544.2, 521.02, 8) mm, rotated rx 180 ry 0 rz 160 deg; joints [8.07, 86.573, -31.115, -147.08, 59.98, 162.052]
  Call Extruder(683.60819)
  MoveL 758 to (543.8, 521.83, 8) mm, rotated rx -180 ry 0 rz 160 deg; joints [8.169, 86.512, -30.981, -146.994, 60.071, 162.043]
  Set speed (17.5 mm/s)
  Call Extruder(688.14909)
  MoveL 759 to (543.16, 523.08, 8) mm, rotated rx 180 ry 0 rz 160 deg; joints [8.322, 86.413, -30.767, -146.863, 60.215, 162.033]
  Set speed (17.5 mm/s)
  Call Extruder(693.28847)
  MoveL 760 to (542.38, 524.47, 8) mm, rotated rx 180 ry 0 rz 160 deg; joints [8.494, 86.292, -30.501, -146.72, 60.388, 162.031]
  Set speed (17.5 mm/s)
  Call Extruder(695.50997)
  MoveL 761 to (542.04, 525.06, 8) mm, rotated rx 180 ry 0 rz 160 deg; joints [8.567, 86.238, -30.383, -146.66, 60.465, 162.032]
  Set speed (17.5 mm/s)
  Call Extruder(701.73365)
  MoveL 762 to (541.01, 526.69, 8) mm, rotated rx 180 ry 0 rz 160 deg; joints [8.771, 86.074, -30.026, -146.497, 60.689, 162.045]
  Set speed (17.5 mm/s)
  Call Extruder(704.56742)
  MoveL 763 to (540.53, 527.42, 8) mm, rotated rx -180 ry 0 rz 160 deg; joints [8.863, 85.997, -29.856, -146.425, 60.795, 162.054]
  Set speed (17.5 mm/s)
  Call Extruder(710.38260)
  MoveL 764 to (539.5, 528.9, 8) mm, rotated rx 180 ry 0 rz 160 deg; joints [9.05, 85.83, -29.49, -146.283, 61.018, 162.081]
  Set speed (17.5 mm/s)
  Call Extruder(715.33513)
  MoveL 765 to (538.57, 530.12, 8) mm, rotated rx 180 ry 0 rz 160 deg; joints [9.207, 85.68, -29.161, -146.168, 61.215, 162.113]
  Call Extruder(719.03529)
  MoveL 766 to (537.86, 531.01, 8) mm, rotated rx 180 ry 0 rz 160 deg; joints [9.323, 85.564, -28.905, -146.085, 61.366, 162.141]
  Call Extruder(722.38087)
  MoveL 767 to (537.19, 531.81, 8) mm, rotated rx 180 ry 0 rz 160 deg; joints [9.426, 85.455, -28.667, -146.012, 61.506, 162.17]
  Call Extruder(727.63317)
  MoveL 768 to (536.11, 533.02, 8) mm, rotated rx 180 ry 0 rz 160 deg; joints [9.586, 85.279, -28.278, -145.903, 61.731, 162.223]
  Set speed (17.5 mm/s)
  Call Extruder(733.54015)
  MoveL 769 to (534.86, 534.35, 8) mm, rotated rx -180 ry 0 rz 160 deg; joints [9.764, 85.073, -27.824, -145.786, 61.99, 162.291]
  Set speed (17.5 mm/s)
  Call Extruder(738.54455)
  MoveL 770 to (533.75, 535.43, 8) mm, rotated rx 180 ry 0 rz 160 deg; joints [9.91, 84.892, -27.423, -145.694, 62.216, 162.357]
  Set speed (17.5 mm/s)
  Call Extruder(742.75060)
  MoveL 771 to (532.8, 536.32, 8) mm, rotated rx -180 ry 0 rz 160 deg; joints [10.032, 84.737, -27.079, -145.618, 62.409, 162.416]
  Call Extruder(745.02414)
  MoveL 772 to (532.27, 536.79, 8) mm, rotated rx -180 ry 0 rz 160 deg; joints [10.096, 84.65, -26.887, -145.58, 62.516, 162.451]
  Set speed (17.5 mm/s)
  Call Extruder(749.79861)
  MoveL 773 to (531.15, 537.75, 8) mm, rotated rx 180 ry 0 rz 160 deg; joints [10.23, 84.467, -26.48, -145.502, 62.741, 162.528]
  Set speed (17.5 mm/s)
  Call Extruder(751.51024)
  MoveL 774 to (530.74, 538.08, 8) mm, rotated rx 180 ry 0 rz 160 deg; joints [10.277, 84.4, -26.33, -145.476, 62.823, 162.557]
  Set speed (17.4 mm/s)
  Call Extruder(757.00131)
  MoveL 775 to (529.4, 539.12, 8) mm, rotated rx 180 ry 0 rz 160 deg; joints [10.426, 84.182, -25.845, -145.393, 63.087, 162.655]
  Set speed (17.4 mm/s)
  Call Extruder(759.33143)
  MoveL 776 to (528.82, 539.55, 8) mm, rotated rx -180 ry 0 rz 160 deg; joints [10.488, 84.088, -25.635, -145.361, 63.201, 162.699]
  Set speed (17.5 mm/s)
  Call Extruder(765.90242)
  MoveL 777 to (527.15, 540.72, 8) mm, rotated rx -180 ry 0 rz 160 deg; joints [10.659, 83.818, -25.031, -145.273, 63.527, 162.83]
  Set speed (17.4 mm/s)
  Call Extruder(767.67985)
  MoveL 778 to (526.69, 541.01, 8) mm, rotated rx 180 ry 0 rz 160 deg; joints [10.704, 83.743, -24.864, -145.252, 63.616, 162.867]
  Set speed (17.4 mm/s)
  Call Extruder(773.49267)
  MoveL 779 to (525.17, 541.97, 8) mm, rotated rx -180 ry 0 rz 160 deg; joints [10.849, 83.498, -24.313, -145.183, 63.909, 162.993]
  Set speed (17.5 mm/s)
  Call Extruder(777.38730)
  MoveL 780 to (524.13, 542.58, 8) mm, rotated rx -180 ry 0 rz 160 deg; joints [10.943, 83.331, -23.937, -145.141, 64.108, 163.082]
  Set speed (17.5 mm/s)
  Call Extruder(780.64202)
  MoveL 781 to (523.25, 543.06, 8) mm, rotated rx -180 ry 0 rz 160 deg; joints [11.02, 83.19, -23.619, -145.109, 64.276, 163.159]
  Set speed (17.4 mm/s)
  Call Extruder(783.87243)
  MoveL 782 to (522.37, 543.53, 8) mm, rotated rx -180 ry 0 rz 160 deg; joints [11.094, 83.049, -23.3, -145.078, 64.443, 163.238]
  Set speed (17.5 mm/s)
  Call Extruder(789.38717)
  MoveL 783 to (520.83, 544.28, 8) mm, rotated rx 180 ry 0 rz 160 deg; joints [11.218, 82.805, -22.749, -145.031, 64.731, 163.377]
  Set speed (17.4 mm/s)
  Call Extruder(793.58602)
  MoveL 784 to (519.65, 544.81, 8) mm, rotated rx 180 ry 0 rz 160 deg; joints [11.308, 82.618, -22.323, -144.999, 64.952, 163.487]
  Set speed (17.4 mm/s)
  Call Extruder(796.72653)
  MoveL 785 to (518.76, 545.2, 8) mm, rotated rx -180 ry 0 rz 160 deg; joints [11.374, 82.478, -22.004, -144.977, 65.117, 163.57]
  Set speed (17.4 mm/s)
  Call Extruder(800.05636)
  MoveL 786 to (517.81, 545.58, 8) mm, rotated rx -180 ry 0 rz 160 deg; joints [11.442, 82.327, -21.661, -144.957, 65.293, 163.662]
  Set speed (17.4 mm/s)
  Call Extruder(803.84151)
  MoveL 787 to (516.71, 545.99, 8) mm, rotated rx -180 ry 0 rz 160 deg; joints [11.517, 82.156, -21.27, -144.935, 65.494, 163.768]
  Set speed (17.4 mm/s)
  Call Extruder(806.58595)
  MoveL 788 to (515.91, 546.27, 8) mm, rotated rx 180 ry 0 rz 160 deg; joints [11.569, 82.031, -20.984, -144.922, 65.641, 163.847]
  Set speed (17.4 mm/s)
  Call Extruder(811.07065)
  MoveL 789 to (514.6, 546.71, 8) mm, rotated rx -180 ry 0 rz 160 deg; joints [11.653, 81.826, -20.514, -144.903, 65.881, 163.978]
  Set speed (17.5 mm/s)
  Call Extruder(813.94093)
  MoveL 790 to (513.75, 546.97, 8) mm, rotated rx 180 ry 0 rz 160 deg; joints [11.704, 81.694, -20.211, -144.892, 66.035, 164.063]
  Call Extruder(818.45640)
  MoveL 791 to (512.4, 547.34, 8) mm, rotated rx 180 ry 0 rz 160 deg; joints [11.782, 81.486, -19.733, -144.88, 66.277, 164.201]
  Set speed (17.4 mm/s)
  Call Extruder(822.71115)
  MoveL 792 to (511.12, 547.65, 8) mm, rotated rx 180 ry 0 rz 160 deg; joints [11.851, 81.289, -19.279, -144.872, 66.506, 164.333]
  Call Extruder(828.64066)
  MoveL 793 to (509.33, 548.04, 8) mm, rotated rx -180 ry 0 rz 160 deg; joints [11.942, 81.015, -18.645, -144.865, 66.826, 164.521]
  Set speed (17.5 mm/s)
  Call Extruder(835.42313)
  MoveL 794 to (507.26, 548.4, 8) mm, rotated rx -180 ry 0 rz 160 deg; joints [12.038, 80.701, -17.914, -144.867, 67.191, 164.742]
  Set speed (17.5 mm/s)
  Call Extruder(842.10961)
  MoveL 795 to (505.21, 548.66, 8) mm, rotated rx -180 ry 0 rz 160 deg; joints [12.122, 80.391, -17.191, -144.878, 67.552, 164.966]
  Set speed (17.4 mm/s)
  Call Extruder(848.62535)
  MoveL 796 to (503.2, 548.83, 8) mm, rotated rx 180 ry 0 rz 160 deg; joints [12.195, 80.091, -16.486, -144.897, 67.901, 165.189]
  Set speed (17.5 mm/s)
  Call Extruder(852.77608)
  MoveL 797 to (501.92, 548.89, 8) mm, rotated rx -180 ry 0 rz 160 deg; joints [12.236, 79.899, -16.035, -144.914, 68.124, 165.333]
  Set speed (17.5 mm/s)
  Call Extruder(855.15676)
  MoveL 798 to (501.18, 548.92, 8) mm, rotated rx 180 ry 0 rz 160 deg; joints [12.259, 79.79, -15.778, -144.925, 68.251, 165.416]
  Set speed (17.4 mm/s)
  Call Extruder(860.83729)
  MoveL 799 to (499.43, 548.93, 8) mm, rotated rx 180 ry 0 rz 160 deg; joints [12.307, 79.531, -15.164, -144.955, 68.553, 165.616]
  Set speed (10.0 mm/s)
  MoveL 800 to (499.43, 548.93, 12) mm, rotated rx -180 ry 0 rz 160 deg; joints [12.307, 78.782, -14.572, -144.92, 68.424, 165.519]
  Set speed (90.0 mm/s)
  MoveL 801 to (499.22, 549.93, 12) mm, rotated rx 180 ry 0 rz 160 deg; joints [12.434, 78.783, -14.577, -144.787, 68.454, 165.469]
  Set speed (17.5 mm/s)
  Call Extruder(867.60571)
  MoveL 802 to (497.13, 549.86, 12) mm, rotated rx 180 ry 0 rz 160 deg; joints [12.481, 78.476, -13.85, -144.833, 68.809, 165.711]
  Set speed (17.5 mm/s)
  Call Extruder(874.22382)
  MoveL 803 to (495.09, 549.7, 12) mm, rotated rx -180 ry 0 rz 160 deg; joints [12.517, 78.179, -13.142, -144.886, 69.153, 165.951]
  Set speed (17.5 mm/s)
  Call Extruder(880.56234)
  MoveL 804 to (493.14, 549.47, 12) mm, rotated rx -180 ry 0 rz 160 deg; joints [12.542, 77.897, -12.468, -144.945, 69.48, 166.182]
  Set speed (17.5 mm/s)
  Call Extruder(887.24535)
  MoveL 805 to (491.1, 549.14, 12) mm, rotated rx 180 ry 0 rz 160 deg; joints [12.558, 77.602, -11.761, -145.017, 69.821, 166.429]
  Set speed (17.5 mm/s)
  Call Extruder(894.04693)
  MoveL 806 to (489.03, 548.72, 12) mm, rotated rx -180 ry 0 rz 160 deg; joints [12.563, 77.307, -11.048, -145.098, 70.165, 166.682]
  Set speed (17.5 mm/s)
  Call Extruder(900.49742)
  MoveL 807 to (487.09, 548.24, 12) mm, rotated rx 180 ry 0 rz 160 deg; joints [12.557, 77.031, -10.379, -145.184, 70.486, 166.922]
  Set speed (17.5 mm/s)
  Call Extruder(907.24606)
  MoveL 808 to (485.09, 547.66, 12) mm, rotated rx 180 ry 0 rz 160 deg; joints [12.54, 76.747, -9.688, -145.283, 70.817, 167.174]
  Set speed (17.4 mm/s)
  Call Extruder(913.60563)
  MoveL 809 to (483.22, 547.04, 12) mm, rotated rx -180 ry 0 rz 160 deg; joints [12.514, 76.485, -9.045, -145.385, 71.124, 167.412]
  Set speed (17.5 mm/s)
  Call Extruder(915.38280)
  MoveL 810 to (482.71, 546.84, 12) mm, rotated rx -180 ry 0 rz 160 deg; joints [12.503, 76.412, -8.867, -145.417, 71.208, 167.479]
  Set speed (17.5 mm/s)
  Call Extruder(916.45914)
  MoveL 811 to (482.4, 546.73, 12) mm, rotated rx -180 ry 0 rz 160 deg; joints [12.498, 76.368, -8.759, -145.434, 71.26, 167.519]
  Set speed (17.4 mm/s)
  Call Extruder(920.47860)
  MoveL 812 to (481.24, 546.28, 12) mm, rotated rx -180 ry 0 rz 160 deg; joints [12.474, 76.206, -8.36, -145.505, 71.45, 167.669]
  Set speed (17.4 mm/s)
  Call Extruder(925.22243)
  MoveL 813 to (479.89, 545.71, 12) mm, rotated rx -180 ry 0 rz 160 deg; joints [12.44, 76.018, -7.894, -145.592, 71.672, 167.845]
  Call Extruder(930.34958)
  MoveL 814 to (478.45, 545.05, 12) mm, rotated rx 180 ry 0 rz 160 deg; joints [12.396, 75.817, -7.397, -145.693, 71.907, 168.036]
  Set speed (17.5 mm/s)
  Call Extruder(933.56321)
  MoveL 815 to (477.56, 544.61, 12) mm, rotated rx -180 ry 0 rz 160 deg; joints [12.364, 75.694, -7.089, -145.759, 72.053, 168.155]
  Set speed (17.5 mm/s)
  Call Extruder(936.82678)
  MoveL 816 to (476.66, 544.15, 12) mm, rotated rx -180 ry 0 rz 160 deg; joints [12.33, 75.569, -6.778, -145.828, 72.2, 168.276]
  Call Extruder(940.07008)
  MoveL 817 to (475.77, 543.67, 12) mm, rotated rx -180 ry 0 rz 160 deg; joints [12.294, 75.447, -6.473, -145.898, 72.344, 168.395]
  Set speed (17.5 mm/s)
  Call Extruder(943.38612)
  MoveL 818 to (474.88, 543.16, 12) mm, rotated rx 180 ry 0 rz 160 deg; joints [12.253, 75.324, -6.164, -145.973, 72.49, 168.517]
  Set speed (17.5 mm/s)
  Call Extruder(946.73714)
  MoveL 819 to (473.99, 542.63, 12) mm, rotated rx -180 ry 0 rz 160 deg; joints [12.209, 75.201, -5.855, -146.05, 72.636, 168.639]
  Call Extruder(950.02551)
  MoveL 820 to (473.13, 542.09, 12) mm, rotated rx -180 ry 0 rz 160 deg; joints [12.164, 75.082, -5.556, -146.128, 72.777, 168.759]
  Call Extruder(953.39588)
  MoveL 821 to (472.25, 541.52, 12) mm, rotated rx 180 ry 0 rz 160 deg; joints [12.114, 74.962, -5.252, -146.211, 72.92, 168.881]
  Set speed (17.5 mm/s)
  Call Extruder(956.62787)
  MoveL 822 to (471.43, 540.96, 12) mm, rotated rx -180 ry 0 rz 160 deg; joints [12.064, 74.849, -4.965, -146.292, 73.055, 168.997]
  Set speed (17.5 mm/s)
  Call Extruder(959.96185)
  MoveL 823 to (470.59, 540.36, 12) mm, rotated rx 180 ry 0 rz 160 deg; joints [12.009, 74.734, -4.673, -146.378, 73.192, 169.116]
  Set speed (17.5 mm/s)
  Call Extruder(963.31377)
  MoveL 824 to (469.76, 539.74, 12) mm, rotated rx -180 ry 0 rz 160 deg; joints [11.951, 74.62, -4.382, -146.467, 73.328, 169.235]
  Set speed (17.5 mm/s)
  Call Extruder(966.56662)
  MoveL 825 to (468.96, 539.12, 12) mm, rotated rx 180 ry 0 rz 160 deg; joints [11.892, 74.511, -4.105, -146.555, 73.458, 169.349]
  Set speed (17.5 mm/s)
  Call Extruder(969.82311)
  MoveL 826 to (468.18, 538.49, 12) mm, rotated rx 180 ry 0 rz 160 deg; joints [11.831, 74.404, -3.83, -146.645, 73.586, 169.463]
  Set speed (17.5 mm/s)
  Call Extruder(973.78126)
  MoveL 827 to (467.24, 537.7, 12) mm, rotated rx -180 ry 0 rz 160 deg; joints [11.752, 74.276, -3.502, -146.758, 73.739, 169.6]
  Set speed (17.5 mm/s)
  Call Extruder(979.63850)
  MoveL 828 to (465.89, 536.48, 12) mm, rotated rx -180 ry 0 rz 160 deg; joints [11.628, 74.092, -3.028, -146.931, 73.96, 169.801]
  Set speed (17.5 mm/s)
  Call Extruder(982.96889)
  MoveL 829 to (465.15, 535.77, 12) mm, rotated rx -180 ry 0 rz 160 deg; joints [11.554, 73.99, -2.765, -147.032, 74.082, 169.913]
  Call Extruder(986.34402)
  MoveL 830 to (464.41, 535.03, 12) mm, rotated rx 180 ry 0 rz 160 deg; joints [11.476, 73.889, -2.503, -147.137, 74.203, 170.026]
  Set speed (17.5 mm/s)
  Call Extruder(989.70425)
  MoveL 831 to (463.69, 534.28, 12) mm, rotated rx 180 ry 0 rz 160 deg; joints [11.396, 73.79, -2.246, -147.243, 74.322, 170.137]
  Set speed (17.5 mm/s)
  Call Extruder(992.89086)
  MoveL 832 to (463.02, 533.56, 12) mm, rotated rx 180 ry 0 rz 160 deg; joints [11.317, 73.698, -2.008, -147.345, 74.432, 170.241]
  Set speed (17.5 mm/s)
  Call Extruder(996.95764)
  MoveL 833 to (462.18, 532.62, 12) mm, rotated rx 180 ry 0 rz 160 deg; joints [11.214, 73.584, -1.709, -147.479, 74.57, 170.372]
  Set speed (17.5 mm/s)
  Call Extruder(1002.78801)
  MoveL 834 to (461.03, 531.23, 12) mm, rotated rx -180 ry 0 rz 160 deg; joints [11.058, 73.426, -1.294, -147.676, 74.761, 170.557]
  Set speed (17.5 mm/s)
  Call Extruder(1006.11215)
  MoveL 835 to (460.39, 530.42, 12) mm, rotated rx 180 ry 0 rz 160 deg; joints [10.965, 73.338, -1.065, -147.791, 74.866, 170.66]
  Set speed (17.5 mm/s)
  Call Extruder(1009.50473)
  MoveL 836 to (459.76, 529.58, 12) mm, rotated rx 180 ry 0 rz 160 deg; joints [10.868, 73.251, -0.836, -147.911, 74.97, 170.764]
  Call Extruder(1012.69362)
  MoveL 837 to (459.19, 528.78, 12) mm, rotated rx -180 ry 0 rz 160 deg; joints [10.775, 73.172, -0.626, -148.025, 75.066, 170.861]
  Set speed (17.5 mm/s)
  Call Extruder(1016.03986)
  MoveL 838 to (458.6, 527.93, 12) mm, rotated rx 180 ry 0 rz 160 deg; joints [10.675, 73.09, -0.411, -148.146, 75.164, 170.96]
  Set speed (17.5 mm/s)
  Call Extruder(1019.32102)
  MoveL 839 to (458.04, 527.08, 12) mm, rotated rx -180 ry 0 rz 160 deg; joints [10.574, 73.013, -0.205, -148.267, 75.257, 171.056]
  Set speed (17.5 mm/s)
  Call Extruder(1022.55518)
  MoveL 840 to (457.5, 526.23, 12) mm, rotated rx 180 ry 0 rz 160 deg; joints [10.472, 72.938, -0.007, -148.388, 75.346, 171.15]
  Set speed (17.5 mm/s)
  Call Extruder(1025.99892)
  MoveL 841 to (456.95, 525.32, 12) mm, rotated rx 180 ry 0 rz 160 deg; joints [10.362, 72.861, 0.199, -148.518, 75.439, 171.248]
  Set speed (17.5 mm/s)
  Call Extruder(1029.28956)
  MoveL 842 to (456.45, 524.43, 12) mm, rotated rx -180 ry 0 rz 160 deg; joints [10.253, 72.79, 0.388, -148.645, 75.523, 171.339]
  Set speed (17.5 mm/s)
  Call Extruder(1034.17162)
  MoveL 843 to (455.73, 523.11, 12) mm, rotated rx -180 ry 0 rz 160 deg; joints [10.089, 72.688, 0.661, -148.835, 75.645, 171.472]
  Call Extruder(1039.21556)
  MoveL 844 to (455.03, 521.71, 12) mm, rotated rx -180 ry 0 rz 160 deg; joints [9.915, 72.588, 0.929, -149.035, 75.763, 171.606]
  Set speed (17.5 mm/s)
  Call Extruder(1045.63374)
  MoveL 845 to (454.2, 519.91, 12) mm, rotated rx 180 ry 0 rz 160 deg; joints [9.686, 72.469, 1.25, -149.295, 75.904, 171.77]
  Set speed (17.4 mm/s)
  Call Extruder(1049.13013)
  MoveL 846 to (453.78, 518.91, 12) mm, rotated rx 180 ry 0 rz 160 deg; joints [9.558, 72.407, 1.416, -149.439, 75.975, 171.856]
  Set speed (17.4 mm/s)
  Call Extruder(1052.40989)
  MoveL 847 to (453.4, 517.97, 12) mm, rotated rx -180 ry 0 rz 160 deg; joints [9.436, 72.351, 1.567, -149.575, 76.04, 171.936]
  Set speed (17.5 mm/s)
  Call Extruder(1059.11167)
  MoveL 848 to (452.7, 516.02, 12) mm, rotated rx -180 ry 0 rz 160 deg; joints [9.182, 72.245, 1.854, -149.857, 76.161, 172.093]
  Call Extruder(1065.40440)
  MoveL 849 to (452.11, 514.16, 12) mm, rotated rx 180 ry 0 rz 160 deg; joints [8.937, 72.154, 2.102, -150.126, 76.263, 172.233]
  Set speed (17.5 mm/s)
  Call Extruder(1072.22403)
  MoveL 850 to (451.55, 512.13, 12) mm, rotated rx 180 ry 0 rz 160 deg; joints [8.665, 72.064, 2.346, -150.422, 76.361, 172.377]
  Set speed (17.5 mm/s)
  Call Extruder(1078.58379)
  MoveL 851 to (451.12, 510.21, 12) mm, rotated rx -180 ry 0 rz 160 deg; joints [8.405, 71.99, 2.549, -150.702, 76.439, 172.504]
  Set speed (17.5 mm/s)
  Call Extruder(1085.44928)
  MoveL 852 to (450.73, 508.12, 12) mm, rotated rx 180 ry 0 rz 160 deg; joints [8.12, 71.92, 2.742, -151.007, 76.509, 172.634]
  Set speed (17.5 mm/s)
  Call Extruder(1092.03502)
  MoveL 853 to (450.43, 506.1, 12) mm, rotated rx -180 ry 0 rz 160 deg; joints [7.843, 71.862, 2.902, -151.302, 76.563, 172.75]
  Call Extruder(1098.63284)
  MoveL 854 to (450.23, 504.07, 12) mm, rotated rx -180 ry 0 rz 160 deg; joints [7.561, 71.813, 3.036, -151.599, 76.602, 172.859]
  Call Extruder(1105.07287)
  MoveL 855 to (450.1, 502.08, 12) mm, rotated rx -180 ry 0 rz 160 deg; joints [7.282, 71.774, 3.142, -151.891, 76.627, 172.957]
  Set speed (17.5 mm/s)
  Call Extruder(1111.75990)
  MoveL 856 to (450.06, 500.01, 12) mm, rotated rx 180 ry 0 rz 160 deg; joints [6.991, 71.744, 3.225, -152.194, 76.639, 173.052]
  Set speed (17.5 mm/s)
  Call Extruder(1117.78136)
  MoveL 857 to (450.09, 498.15, 12) mm, rotated rx -180 ry 0 rz 160 deg; joints [6.727, 71.725, 3.279, -152.467, 76.637, 173.13]
  Set speed (17.5 mm/s)
  Call Extruder(1123.63199)
  MoveL 858 to (450.19, 496.34, 12) mm, rotated rx 180 ry 0 rz 160 deg; joints [6.47, 71.714, 3.309, -152.732, 76.624, 173.2]
  Call Extruder(1129.52489)
  MoveL 859 to (450.36, 494.53, 12) mm, rotated rx 180 ry 0 rz 160 deg; joints [6.21, 71.71, 3.318, -152.998, 76.598, 173.264]
  Call Extruder(1135.43774)
  MoveL 860 to (450.6, 492.71, 12) mm, rotated rx 180 ry 0 rz 160 deg; joints [5.949, 71.714, 3.307, -153.264, 76.561, 173.323]
  Call Extruder(1141.54575)
  MoveL 861 to (450.91, 490.85, 12) mm, rotated rx 180 ry 0 rz 160 deg; joints [5.68, 71.726, 3.274, -153.536, 76.511, 173.377]
  Call Extruder(1147.34823)
  MoveL 862 to (451.27, 489.09, 12) mm, rotated rx -180 ry 0 rz 160 deg; joints [5.426, 71.746, 3.221, -153.792, 76.452, 173.422]
  Set speed (17.5 mm/s)
  Call Extruder(1153.34594)
  MoveL 863 to (451.71, 487.28, 12) mm, rotated rx 180 ry 0 rz 160 deg; joints [5.164, 71.773, 3.145, -154.054, 76.379, 173.463]
  Call Extruder(1159.16681)
  MoveL 864 to (452.2, 485.55, 12) mm, rotated rx 180 ry 0 rz 160 deg; joints [4.912, 71.807, 3.051, -154.305, 76.296, 173.497]
  Set speed (17.5 mm/s)
  Call Extruder(1165.14530)
  MoveL 865 to (452.76, 483.79, 12) mm, rotated rx -180 ry 0 rz 160 deg; joints [4.656, 71.85, 2.933, -154.56, 76.2, 173.526]
  Call Extruder(1171.19649)
  MoveL 866 to (453.41, 482.03, 12) mm, rotated rx -180 ry 0 rz 160 deg; joints [4.4, 71.901, 2.792, -154.812, 76.09, 173.55]
  Call Extruder(1177.19048)
  MoveL 867 to (454.11, 480.31, 12) mm, rotated rx -180 ry 0 rz 160 deg; joints [4.15, 71.96, 2.632, -155.058, 75.97, 173.567]
  Set speed (17.5 mm/s)
  Call Extruder(1182.94819)
  MoveL 868 to (454.84, 478.69, 12) mm, rotated rx 180 ry 0 rz 160 deg; joints [3.913, 72.023, 2.459, -155.289, 75.844, 173.579]
  Call Extruder(1189.06933)
  MoveL 869 to (455.68, 476.99, 12) mm, rotated rx 180 ry 0 rz 160 deg; joints [3.666, 72.098, 2.254, -155.529, 75.698, 173.585]
  Set speed (17.5 mm/s)
  Call Extruder(1194.90796)
  MoveL 870 to (456.54, 475.4, 12) mm, rotated rx -180 ry 0 rz 160 deg; joints [3.434, 72.178, 2.038, -155.751, 75.547, 173.586]
  Call Extruder(1200.84757)
  MoveL 871 to (457.48, 473.81, 12) mm, rotated rx 180 ry 0 rz 160 deg; joints [3.204, 72.266, 1.799, -155.972, 75.384, 173.581]
  Call Extruder(1206.78750)
  MoveL 872 to (458.47, 472.27, 12) mm, rotated rx 180 ry 0 rz 160 deg; joints [2.98, 72.361, 1.54, -156.185, 75.21, 173.571]
  Set speed (17.5 mm/s)
  Call Extruder(1212.72915)
  MoveL 873 to (459.52, 470.76, 12) mm, rotated rx -180 ry 0 rz 160 deg; joints [2.761, 72.464, 1.262, -156.391, 75.025, 173.556]
  Set speed (17.5 mm/s)
  Call Extruder(1218.75267)
  MoveL 874 to (460.64, 469.26, 12) mm, rotated rx 180 ry 0 rz 160 deg; joints [2.545, 72.576, 0.962, -156.593, 74.827, 173.536]
  Set speed (17.5 mm/s)
  Call Extruder(1224.53794)
  MoveL 875 to (461.77, 467.87, 12) mm, rotated rx 180 ry 0 rz 160 deg; joints [2.345, 72.69, 0.654, -156.779, 74.628, 173.511]
  Set speed (17.5 mm/s)
  Call Extruder(1230.54789)
  MoveL 876 to (462.99, 466.47, 12) mm, rotated rx -180 ry 0 rz 160 deg; joints [2.143, 72.817, 0.317, -156.963, 74.411, 173.481]
  Set speed (17.5 mm/s)
  Call Extruder(1236.56394)
  MoveL 877 to (464.27, 465.12, 12) mm, rotated rx 180 ry 0 rz 160 deg; joints [1.949, 72.95, -0.039, -157.139, 74.184, 173.445]
  Set speed (17.5 mm/s)
  Call Extruder(1242.42427)
  MoveL 878 to (465.56, 463.84, 12) mm, rotated rx 180 ry 0 rz 160 deg; joints [1.767, 73.087, -0.403, -157.302, 73.954, 173.405]
  Set speed (17.5 mm/s)
  Call Extruder(1248.36404)
  MoveL 879 to (466.91, 462.6, 12) mm, rotated rx 180 ry 0 rz 160 deg; joints [1.59, 73.233, -0.789, -157.459, 73.712, 173.36]
  Set speed (17.5 mm/s)
  Call Extruder(1254.38523)
  MoveL 880 to (468.33, 461.39, 12) mm, rotated rx -180 ry 0 rz 160 deg; joints [1.419, 73.388, -1.197, -157.607, 73.458, 173.309]
  Call Extruder(1260.16605)
  MoveL 881 to (469.73, 460.28, 12) mm, rotated rx 180 ry 0 rz 160 deg; joints [1.263, 73.544, -1.604, -157.741, 73.207, 173.256]
  Set speed (17.5 mm/s)
  Call Extruder(1266.22010)
  MoveL 882 to (471.24, 459.17, 12) mm, rotated rx -180 ry 0 rz 160 deg; joints [1.107, 73.713, -2.046, -157.871, 72.936, 173.195]
  Call Extruder(1272.01343)
  MoveL 883 to (472.73, 458.17, 12) mm, rotated rx -180 ry 0 rz 160 deg; joints [0.967, 73.882, -2.485, -157.985, 72.669, 173.132]
  Call Extruder(1278.14244)
  MoveL 884 to (474.34, 457.16, 12) mm, rotated rx -180 ry 0 rz 160 deg; joints [0.827, 74.067, -2.964, -158.096, 72.38, 173.061]
  Set speed (17.5 mm/s)
  Call Extruder(1284.07048)
  MoveL 885 to (475.93, 456.25, 12) mm, rotated rx -180 ry 0 rz 160 deg; joints [0.701, 74.252, -3.442, -158.192, 72.093, 172.986]
  Set speed (17.4 mm/s)
  Call Extruder(1290.88250)
  MoveL 886 to (477.79, 455.27, 12) mm, rotated rx 180 ry 0 rz 160 deg; joints [0.567, 74.473, -4.007, -158.291, 71.757, 172.895]
  Set speed (17.4 mm/s)
  Call Extruder(1295.97485)
  MoveL 887 to (479.22, 454.59, 12) mm, rotated rx -180 ry 0 rz 160 deg; joints [0.475, 74.643, -4.441, -158.355, 71.499, 172.823]
  Set speed (17.5 mm/s)
  Call Extruder(1301.91907)
  MoveL 888 to (480.9, 453.86, 12) mm, rotated rx -180 ry 0 rz 160 deg; joints [0.375, 74.847, -4.96, -158.421, 71.194, 172.734]
  Set speed (17.5 mm/s)
  Call Extruder(1307.68328)
  MoveL 889 to (482.56, 453.2, 12) mm, rotated rx 180 ry 0 rz 160 deg; joints [0.287, 75.05, -5.475, -158.473, 70.893, 172.643]
  Set speed (17.5 mm/s)
  Call Extruder(1313.78883)
  MoveL 890 to (484.35, 452.58, 12) mm, rotated rx 180 ry 0 rz 160 deg; joints [0.203, 75.271, -6.032, -158.519, 70.57, 172.542]
  Set speed (17.5 mm/s)
  Call Extruder(1319.57290)
  MoveL 891 to (486.06, 452.05, 12) mm, rotated rx 180 ry 0 rz 160 deg; joints [0.132, 75.486, -6.571, -158.551, 70.259, 172.441]
  Set speed (17.5 mm/s)
  Call Extruder(1325.43120)
  MoveL 892 to (487.81, 451.57, 12) mm, rotated rx 180 ry 0 rz 160 deg; joints [0.069, 75.709, -7.126, -158.573, 69.941, 172.334]
  Call Extruder(1331.60019)
  MoveL 893 to (489.67, 451.14, 12) mm, rotated rx -180 ry 0 rz 160 deg; joints [0.013, 75.948, -7.722, -158.584, 69.602, 172.216]
  Set speed (17.5 mm/s)
  Call Extruder(1337.45300)
  MoveL 894 to (491.45, 450.8, 12) mm, rotated rx -180 ry 0 rz 160 deg; joints [-0.032, 76.18, -8.296, -158.585, 69.277, 172.099]
  Set speed (17.5 mm/s)
  Call Extruder(1343.25906)
  MoveL 895 to (493.23, 450.52, 12) mm, rotated rx 180 ry 0 rz 160 deg; joints [-0.067, 76.415, -8.874, -158.575, 68.953, 171.978]
  Set speed (17.5 mm/s)
  Call Extruder(1349.32274)
  MoveL 896 to (495.09, 450.3, 12) mm, rotated rx -180 ry 0 rz 160 deg; joints [-0.095, 76.664, -9.485, -158.553, 68.612, 171.847]
  Set speed (17.5 mm/s)
  Call Extruder(1355.20366)
  MoveL 897 to (496.9, 450.16, 12) mm, rotated rx -180 ry 0 rz 160 deg; joints [-0.114, 76.91, -10.085, -158.521, 68.28, 171.715]
  Set speed (17.5 mm/s)
  Call Extruder(1361.29359)
  MoveL 898 to (498.79, 450.08, 12) mm, rotated rx -180 ry 0 rz 160 deg; joints [-0.124, 77.169, -10.713, -158.478, 67.934, 171.573]
  Set speed (17.5 mm/s)
  Call Extruder(1367.16544)
  MoveL 899 to (500.6, 450.06, 12) mm, rotated rx 180 ry 0 rz 160 deg; joints [-0.125, 77.422, -11.325, -158.425, 67.6, 171.431]
  Set speed (17.5 mm/s)
  Call Extruder(1372.99912)
  MoveL 900 to (502.41, 450.12, 12) mm, rotated rx 180 ry 0 rz 160 deg; joints [-0.117, 77.676, -11.938, -158.362, 67.268, 171.285]
  Set speed (17.5 mm/s)
  Call Extruder(1379.03829)
  MoveL 901 to (504.27, 450.24, 12) mm, rotated rx -180 ry 0 rz 160 deg; joints [-0.101, 77.943, -12.578, -158.286, 66.924, 171.129]
  Set speed (17.5 mm/s)
  Call Extruder(1385.04054)
  MoveL 902 to (506.12, 450.44, 12) mm, rotated rx -180 ry 0 rz 160 deg; joints [-0.076, 78.21, -13.217, -158.201, 66.583, 170.968]
  Set speed (17.5 mm/s)
  Call Extruder(1390.86373)
  MoveL 903 to (507.91, 450.69, 12) mm, rotated rx 180 ry 0 rz 160 deg; joints [-0.044, 78.472, -13.84, -158.107, 66.253, 170.808]
  Call Extruder(1396.68841)
  MoveL 904 to (509.68, 451.01, 12) mm, rotated rx -180 ry 0 rz 160 deg; joints [-0.004, 78.736, -14.465, -158.005, 65.924, 170.643]
  Call Extruder(1402.68052)
  MoveL 905 to (511.49, 451.4, 12) mm, rotated rx -180 ry 0 rz 160 deg; joints [0.045, 79.01, -15.111, -157.889, 65.588, 170.468]
  Set speed (17.5 mm/s)
  Call Extruder(1408.73539)
  MoveL 906 to (513.31, 451.87, 12) mm, rotated rx 180 ry 0 rz 160 deg; joints [0.102, 79.288, -15.764, -157.762, 65.25, 170.286]
  Call Extruder(1414.66259)
  MoveL 907 to (515.07, 452.39, 12) mm, rotated rx 180 ry 0 rz 160 deg; joints [0.166, 79.561, -16.403, -157.628, 64.922, 170.104]
  Call Extruder(1420.68361)
  MoveL 908 to (516.84, 452.99, 12) mm, rotated rx 180 ry 0 rz 160 deg; joints [0.239, 79.839, -17.052, -157.482, 64.592, 169.914]
  Set speed (17.5 mm/s)
  Call Extruder(1426.54438)
  MoveL 909 to (518.53, 453.63, 12) mm, rotated rx 180 ry 0 rz 160 deg; joints [0.316, 80.111, -17.682, -157.331, 64.275, 169.724]
  Set speed (17.5 mm/s)
  Call Extruder(1432.57121)
  MoveL 910 to (520.25, 454.35, 12) mm, rotated rx 180 ry 0 rz 160 deg; joints [0.404, 80.39, -18.328, -157.167, 63.952, 169.525]
  Set speed (17.5 mm/s)
  Call Extruder(1438.40578)
  MoveL 911 to (521.89, 455.11, 12) mm, rotated rx -180 ry 0 rz 160 deg; joints [0.495, 80.66, -18.95, -156.999, 63.645, 169.328]
  Set speed (17.5 mm/s)
  Call Extruder(1444.43783)
  MoveL 912 to (523.55, 455.96, 12) mm, rotated rx -180 ry 0 rz 160 deg; joints [0.596, 80.938, -19.589, -156.818, 63.332, 169.12]
  Set speed (17.5 mm/s)
  Call Extruder(1450.37898)
  MoveL 913 to (525.16, 456.86, 12) mm, rotated rx 180 ry 0 rz 160 deg; joints [0.703, 81.211, -20.213, -156.63, 63.029, 168.912]
  Set speed (17.5 mm/s)
  Call Extruder(1456.22777)
  MoveL 914 to (526.71, 457.8, 12) mm, rotated rx 180 ry 0 rz 160 deg; joints [0.814, 81.477, -20.822, -156.439, 62.737, 168.703]
  Call Extruder(1462.24981)
  MoveL 915 to (528.26, 458.83, 12) mm, rotated rx 180 ry 0 rz 160 deg; joints [0.934, 81.75, -21.442, -156.233, 62.443, 168.485]
  Call Extruder(1468.10991)
  MoveL 916 to (529.74, 459.88, 12) mm, rotated rx -180 ry 0 rz 160 deg; joints [1.057, 82.013, -22.037, -156.026, 62.163, 168.269]
  Set speed (17.5 mm/s)
  Call Extruder(1474.05104)
  MoveL 917 to (531.19, 461, 12) mm, rotated rx -180 ry 0 rz 160 deg; joints [1.188, 82.277, -22.634, -155.81, 61.887, 168.048]
  Set speed (17.5 mm/s)
  Call Extruder(1479.98777)
  MoveL 918 to (532.61, 462.18, 12) mm, rotated rx -180 ry 0 rz 160 deg; joints [1.324, 82.537, -23.22, -155.587, 61.618, 167.824]
  Set speed (17.5 mm/s)
  Call Extruder(1486.14479)
  MoveL 919 to (534.03, 463.45, 12) mm, rotated rx -180 ry 0 rz 160 deg; joints [1.471, 82.803, -23.816, -155.348, 61.348, 167.59]
  Call Extruder(1491.90789)
  MoveL 920 to (535.31, 464.69, 12) mm, rotated rx -180 ry 0 rz 160 deg; joints [1.613, 83.048, -24.365, -155.12, 61.103, 167.369]
  Set speed (17.5 mm/s)
  Call Extruder(1495.17918)
  MoveL 921 to (536.02, 465.41, 12) mm, rotated rx -180 ry 0 rz 160 deg; joints [1.696, 83.184, -24.67, -154.988, 60.969, 167.242]
  Call Extruder(1498.46975)
  MoveL 922 to (536.72, 466.15, 12) mm, rotated rx 180 ry 0 rz 160 deg; joints [1.781, 83.32, -24.974, -154.854, 60.836, 167.115]
  Set speed (17.5 mm/s)
  Call Extruder(1501.74387)
  MoveL 923 to (537.4, 466.91, 12) mm, rotated rx -180 ry 0 rz 160 deg; joints [1.867, 83.454, -25.271, -154.719, 60.706, 166.988]
  Set speed (17.5 mm/s)
  Call Extruder(1504.98366)
  MoveL 924 to (538.06, 467.67, 12) mm, rotated rx 180 ry 0 rz 160 deg; joints [1.953, 83.585, -25.562, -154.583, 60.582, 166.862]
  Set speed (17.5 mm/s)
  Call Extruder(1508.33266)
  MoveL 925 to (538.72, 468.46, 12) mm, rotated rx 180 ry 0 rz 160 deg; joints [2.044, 83.718, -25.858, -154.442, 60.455, 166.732]
  Set speed (17.5 mm/s)
  Call Extruder(1511.59163)
  MoveL 926 to (539.35, 469.25, 12) mm, rotated rx -180 ry 0 rz 160 deg; joints [2.134, 83.845, -26.141, -154.304, 60.336, 166.605]
  Set speed (17.5 mm/s)
  Call Extruder(1514.89903)
  MoveL 927 to (539.97, 470.07, 12) mm, rotated rx -180 ry 0 rz 160 deg; joints [2.227, 83.973, -26.423, -154.162, 60.218, 166.476]
  Set speed (17.5 mm/s)
  Call Extruder(1517.61592)
  MoveL 928 to (540.47, 470.74, 12) mm, rotated rx -180 ry 0 rz 160 deg; joints [2.303, 84.076, -26.652, -154.044, 60.123, 166.37]
  Call Extruder(1521.46363)
  MoveL 929 to (541.15, 471.71, 12) mm, rotated rx 180 ry 0 rz 160 deg; joints [2.413, 84.219, -26.968, -153.877, 59.994, 166.22]
  Set speed (17.5 mm/s)
  Call Extruder(1524.76207)
  MoveL 930 to (541.73, 472.56, 12) mm, rotated rx 180 ry 0 rz 160 deg; joints [2.509, 84.34, -27.235, -153.732, 59.885, 166.092]
  Set speed (17.5 mm/s)
  Call Extruder(1528.13824)
  MoveL 931 to (542.29, 473.44, 12) mm, rotated rx 180 ry 0 rz 160 deg; joints [2.609, 84.461, -27.502, -153.583, 59.779, 165.961]
  Set speed (17.5 mm/s)
  Call Extruder(1531.40202)
  MoveL 932 to (542.82, 474.3, 12) mm, rotated rx -180 ry 0 rz 160 deg; joints [2.706, 84.576, -27.754, -153.438, 59.68, 165.835]
  Set speed (17.5 mm/s)
  Call Extruder(1534.67252)
  MoveL 933 to (543.33, 475.17, 12) mm, rotated rx -180 ry 0 rz 160 deg; joints [2.804, 84.688, -28.002, -153.292, 59.583, 165.709]
  Set speed (17.5 mm/s)
  Call Extruder(1538.01072)
  MoveL 934 to (543.83, 476.07, 12) mm, rotated rx 180 ry 0 rz 160 deg; joints [2.906, 84.8, -28.248, -153.142, 59.489, 165.581]
  Set speed (17.5 mm/s)
  Call Extruder(1541.26962)
  MoveL 935 to (544.31, 476.97, 12) mm, rotated rx -180 ry 0 rz 160 deg; joints [3.006, 84.907, -28.482, -152.995, 59.4, 165.457]
  Set speed (17.5 mm/s)
  Call Extruder(1544.62289)
  MoveL 936 to (544.78, 477.89, 12) mm, rotated rx -180 ry 0 rz 160 deg; joints [3.111, 85.014, -28.716, -152.843, 59.313, 165.329]
  Set speed (17.5 mm/s)
  Call Extruder(1547.94032)
  MoveL 937 to (545.22, 478.82, 12) mm, rotated rx 180 ry 0 rz 160 deg; joints [3.215, 85.116, -28.941, -152.693, 59.23, 165.204]
  Set speed (17.5 mm/s)
  Call Extruder(1551.23558)
  MoveL 938 to (545.65, 479.75, 12) mm, rotated rx 180 ry 0 rz 160 deg; joints [3.319, 85.216, -29.159, -152.543, 59.152, 165.081]
  Call Extruder(1557.89863)
  MoveL 939 to (546.44, 481.65, 12) mm, rotated rx 180 ry 0 rz 160 deg; joints [3.533, 85.408, -29.578, -152.24, 59.006, 164.835]
  Set speed (17.5 mm/s)
  Call Extruder(1564.33601)
  MoveL 940 to (547.14, 483.52, 12) mm, rotated rx 180 ry 0 rz 160 deg; joints [3.743, 85.58, -29.955, -151.946, 58.881, 164.601]
  Set speed (17.5 mm/s)
  Call Extruder(1567.77786)
  MoveL 941 to (547.48, 484.53, 12) mm, rotated rx -180 ry 0 rz 160 deg; joints [3.856, 85.667, -30.142, -151.789, 58.822, 164.479]
  Call Extruder(0.00000)
  Call Extruder(3.46971)
  MoveL 942 to (547.8, 485.55, 12) mm, rotated rx -180 ry 0 rz 160 deg; joints [3.971, 85.752, -30.328, -151.631, 58.765, 164.357]
  Set speed (17.5 mm/s)
  Call Extruder(9.69086)
  MoveL 943 to (548.32, 487.4, 12) mm, rotated rx 180 ry 0 rz 160 deg; joints [4.179, 85.893, -30.634, -151.349, 58.676, 164.143]
  Set speed (17.5 mm/s)
  Call Extruder(13.19962)
  MoveL 944 to (548.58, 488.46, 12) mm, rotated rx -180 ry 0 rz 160 deg; joints [4.298, 85.966, -30.793, -151.19, 58.633, 164.025]
  Set speed (17.5 mm/s)
  Call Extruder(16.39917)
  MoveL 945 to (548.8, 489.42, 12) mm, rotated rx -180 ry 0 rz 160 deg; joints [4.406, 86.031, -30.934, -151.046, 58.597, 163.919]
  Set speed (17.5 mm/s)
  Call Extruder(23.07982)
  MoveL 946 to (549.2, 491.45, 12) mm, rotated rx 180 ry 0 rz 160 deg; joints [4.634, 86.153, -31.199, -150.746, 58.536, 163.703]
  Set speed (17.5 mm/s)
  Call Extruder(29.67505)
  MoveL 947 to (549.51, 493.47, 12) mm, rotated rx -180 ry 0 rz 160 deg; joints [4.862, 86.257, -31.425, -150.454, 58.494, 163.499]
  Call Extruder(36.37196)
  MoveL 948 to (549.74, 495.53, 12) mm, rotated rx 180 ry 0 rz 160 deg; joints [5.094, 86.348, -31.621, -150.16, 58.468, 163.301]
  Call Extruder(42.86917)
  MoveL 949 to (549.88, 497.53, 12) mm, rotated rx 180 ry 0 rz 160 deg; joints [5.321, 86.42, -31.776, -149.88, 58.462, 163.119]
  Set speed (17.5 mm/s)
  Call Extruder(49.47476)
  MoveL 950 to (549.94, 499.58, 12) mm, rotated rx -180 ry 0 rz 160 deg; joints [5.553, 86.476, -31.898, -149.599, 58.473, 162.944]
  Set speed (17.5 mm/s)
  Call Extruder(55.95411)
  MoveL 951 to (549.91, 501.58, 12) mm, rotated rx -180 ry 0 rz 160 deg; joints [5.781, 86.515, -31.983, -149.329, 58.501, 162.783]
  Set speed (17.5 mm/s)
  Call Extruder(62.65964)
  MoveL 952 to (549.81, 503.66, 12) mm, rotated rx -180 ry 0 rz 160 deg; joints [6.018, 86.539, -32.035, -149.056, 58.547, 162.628]
  Set speed (17.5 mm/s)
  Call Extruder(69.17721)
  MoveL 953 to (549.62, 505.67, 12) mm, rotated rx -180 ry 0 rz 160 deg; joints [6.248, 86.545, -32.047, -148.796, 58.61, 162.49]
  Set speed (17.5 mm/s)
  Call Extruder(75.95993)
  MoveL 954 to (549.34, 507.75, 12) mm, rotated rx 180 ry 0 rz 160 deg; joints [6.488, 86.534, -32.024, -148.532, 58.694, 162.358]
  Set speed (17.5 mm/s)
  Call Extruder(82.45968)
  MoveL 955 to (548.98, 509.73, 12) mm, rotated rx -180 ry 0 rz 160 deg; joints [6.718, 86.507, -31.965, -148.287, 58.79, 162.245]
  Set speed (17.5 mm/s)
  Call Extruder(88.88873)
  MoveL 956 to (548.56, 511.67, 12) mm, rotated rx 180 ry 0 rz 160 deg; joints [6.944, 86.464, -31.871, -148.051, 58.902, 162.146]
  Set speed (17.5 mm/s)
  Call Extruder(92.38517)
  MoveL 957 to (548.29, 512.72, 12) mm, rotated rx 180 ry 0 rz 160 deg; joints [7.066, 86.433, -31.804, -147.926, 58.97, 162.098]
  Set speed (17.5 mm/s)
  Call Extruder(95.84932)
  MoveL 958 to (548.01, 513.76, 12) mm, rotated rx -180 ry 0 rz 160 deg; joints [7.188, 86.399, -31.732, -147.804, 59.041, 162.053]
  Set speed (17.5 mm/s)
  Call Extruder(102.14833)
  MoveL 959 to (547.43, 515.62, 12) mm, rotated rx -180 ry 0 rz 160 deg; joints [7.408, 86.325, -31.571, -147.588, 59.182, 161.981]
  Set speed (17.5 mm/s)
  Call Extruder(108.75129)
  MoveL 960 to (546.75, 517.55, 12) mm, rotated rx 180 ry 0 rz 160 deg; joints [7.636, 86.231, -31.369, -147.37, 59.344, 161.92]
  Set speed (17.5 mm/s)
  Call Extruder(115.57456)
  MoveL 961 to (545.97, 519.51, 12) mm, rotated rx 180 ry 0 rz 160 deg; joints [7.871, 86.119, -31.125, -147.152, 59.528, 161.871]
  Set speed (17.5 mm/s)
  Call Extruder(121.98309)
  MoveL 962 to (545.16, 521.32, 12) mm, rotated rx -180 ry 0 rz 160 deg; joints [8.09, 85.997, -30.861, -146.957, 59.715, 161.839]
  Set speed (17.5 mm/s)
  Call Extruder(125.27007)
  MoveL 963 to (544.71, 522.24, 12) mm, rotated rx -180 ry 0 rz 160 deg; joints [8.201, 85.929, -30.713, -146.86, 59.817, 161.828]
  Call Extruder(128.67826)
  MoveL 964 to (544.24, 523.18, 12) mm, rotated rx 180 ry 0 rz 160 deg; joints [8.316, 85.856, -30.554, -146.761, 59.925, 161.819]
  Set speed (17.5 mm/s)
  Call Extruder(131.93953)
  MoveL 965 to (543.76, 524.07, 12) mm, rotated rx -180 ry 0 rz 160 deg; joints [8.425, 85.781, -30.392, -146.669, 60.032, 161.814]
  Set speed (17.5 mm/s)
  Call Extruder(135.23006)
  MoveL 966 to (543.26, 524.95, 12) mm, rotated rx 180 ry 0 rz 160 deg; joints [8.534, 85.703, -30.222, -146.579, 60.143, 161.813]
  Set speed (17.5 mm/s)
  Call Extruder(138.46894)
  MoveL 967 to (542.75, 525.82, 12) mm, rotated rx -180 ry 0 rz 160 deg; joints [8.641, 85.622, -30.046, -146.492, 60.255, 161.815]
  Set speed (17.5 mm/s)
  Call Extruder(141.20967)
  MoveL 968 to (542.3, 526.54, 12) mm, rotated rx 180 ry 0 rz 160 deg; joints [8.731, 85.552, -29.893, -146.419, 60.352, 161.819]
  Call Extruder(145.08201)
  MoveL 969 to (541.65, 527.55, 12) mm, rotated rx -180 ry 0 rz 160 deg; joints [8.857, 85.448, -29.667, -146.32, 60.494, 161.829]
  Set speed (17.5 mm/s)
  Call Extruder(148.45765)
  MoveL 970 to (541.07, 528.41, 12) mm, rotated rx -180 ry 0 rz 160 deg; joints [8.966, 85.354, -29.461, -146.236, 60.621, 161.842]
  Set speed (17.5 mm/s)
  Call Extruder(151.72812)
  MoveL 971 to (540.48, 529.24, 12) mm, rotated rx 180 ry 0 rz 160 deg; joints [9.071, 85.26, -29.255, -146.156, 60.746, 161.857]
  Set speed (17.5 mm/s)
  Call Extruder(154.95291)
  MoveL 972 to (539.89, 530.04, 12) mm, rotated rx 180 ry 0 rz 160 deg; joints [9.174, 85.164, -29.046, -146.08, 60.872, 161.875]
  Call Extruder(158.28046)
  MoveL 973 to (539.26, 530.86, 12) mm, rotated rx 180 ry 0 rz 160 deg; joints [9.279, 85.062, -28.823, -146.003, 61.005, 161.897]
  Call Extruder(161.58367)
  MoveL 974 to (538.62, 531.66, 12) mm, rotated rx 180 ry 0 rz 160 deg; joints [9.382, 84.958, -28.595, -145.93, 61.14, 161.922]
  Set speed (17.5 mm/s)
  Call Extruder(164.98580)
  MoveL 975 to (537.95, 532.47, 12) mm, rotated rx 180 ry 0 rz 160 deg; joints [9.487, 84.848, -28.353, -145.856, 61.282, 161.951]
  Set speed (17.5 mm/s)
  Call Extruder(168.19949)
  MoveL 976 to (537.29, 533.21, 12) mm, rotated rx 180 ry 0 rz 160 deg; joints [9.586, 84.741, -28.118, -145.789, 61.418, 161.982]
  Call Extruder(171.46264)
  MoveL 977 to (536.61, 533.96, 12) mm, rotated rx 180 ry 0 rz 160 deg; joints [9.684, 84.63, -27.875, -145.723, 61.558, 162.016]
  Set speed (17.5 mm/s)
  Call Extruder(174.76977)
  MoveL 978 to (535.91, 534.71, 12) mm, rotated rx -180 ry 0 rz 160 deg; joints [9.783, 84.515, -27.622, -145.658, 61.703, 162.053]
  Set speed (17.5 mm/s)
  Call Extruder(178.05231)
  MoveL 979 to (535.2, 535.43, 12) mm, rotated rx 180 ry 0 rz 160 deg; joints [9.881, 84.399, -27.365, -145.595, 61.848, 162.094]
  Set speed (17.5 mm/s)
  Call Extruder(181.45263)
  MoveL 980 to (534.44, 536.16, 12) mm, rotated rx -180 ry 0 rz 160 deg; joints [9.98, 84.275, -27.093, -145.533, 62.002, 162.139]
  Set speed (17.5 mm/s)
  Call Extruder(184.67244)
  MoveL 981 to (533.71, 536.84, 12) mm, rotated rx 180 ry 0 rz 160 deg; joints [10.073, 84.156, -26.83, -145.476, 62.149, 162.184]
  Set speed (17.5 mm/s)
  Call Extruder(187.97594)
  MoveL 982 to (532.95, 537.52, 12) mm, rotated rx -180 ry 0 rz 160 deg; joints [10.167, 84.032, -26.555, -145.42, 62.302, 162.233]
  Set speed (17.5 mm/s)
  Call Extruder(191.29139)
  MoveL 983 to (532.17, 538.2, 12) mm, rotated rx 180 ry 0 rz 160 deg; joints [10.261, 83.906, -26.275, -145.365, 62.456, 162.285]
  Set speed (17.5 mm/s)
  Call Extruder(194.99389)
  MoveL 984 to (531.29, 538.92, 12) mm, rotated rx 180 ry 0 rz 160 deg; joints [10.363, 83.762, -25.955, -145.306, 62.632, 162.347]
  Set speed (17.4 mm/s)
  Call Extruder(199.73349)
  MoveL 985 to (530.13, 539.83, 12) mm, rotated rx 180 ry 0 rz 160 deg; joints [10.492, 83.574, -25.538, -145.236, 62.859, 162.431]
  Set speed (17.4 mm/s)
  Call Extruder(204.55757)
  MoveL 986 to (528.93, 540.71, 12) mm, rotated rx 180 ry 0 rz 160 deg; joints [10.62, 83.379, -25.103, -145.169, 63.094, 162.522]
  Set speed (17.5 mm/s)
  Call Extruder(207.78689)
  MoveL 987 to (528.11, 541.28, 12) mm, rotated rx 180 ry 0 rz 160 deg; joints [10.704, 83.246, -24.807, -145.126, 63.254, 162.586]
  Set speed (17.5 mm/s)
  Call Extruder(211.11037)
  MoveL 988 to (527.25, 541.85, 12) mm, rotated rx 180 ry 0 rz 160 deg; joints [10.788, 83.107, -24.499, -145.084, 63.419, 162.654]
  Call Extruder(214.39521)
  MoveL 989 to (526.39, 542.39, 12) mm, rotated rx 180 ry 0 rz 160 deg; joints [10.871, 82.969, -24.189, -145.045, 63.583, 162.725]
  Set speed (17.5 mm/s)
  Call Extruder(217.64967)
  MoveL 990 to (525.54, 542.92, 12) mm, rotated rx -180 ry 0 rz 160 deg; joints [10.951, 82.831, -23.88, -145.008, 63.747, 162.796]
  Set speed (17.5 mm/s)
  Call Extruder(220.97578)
  MoveL 991 to (524.64, 543.43, 12) mm, rotated rx 180 ry 0 rz 160 deg; joints [11.031, 82.688, -23.56, -144.973, 63.917, 162.872]
  Set speed (17.5 mm/s)
  Call Extruder(224.47541)
  MoveL 992 to (523.7, 543.96, 12) mm, rotated rx 180 ry 0 rz 160 deg; joints [11.114, 82.537, -23.22, -144.938, 64.095, 162.954]
  Set speed (17.5 mm/s)
  Call Extruder(229.55177)
  MoveL 993 to (522.3, 544.68, 12) mm, rotated rx -180 ry 0 rz 160 deg; joints [11.231, 82.315, -22.72, -144.891, 64.357, 163.077]
  Set speed (17.4 mm/s)
  Call Extruder(234.14403)
  MoveL 994 to (521.02, 545.3, 12) mm, rotated rx 180 ry 0 rz 160 deg; joints [11.333, 82.112, -22.262, -144.853, 64.595, 163.194]
  Set speed (17.4 mm/s)
  Call Extruder(239.33509)
  MoveL 995 to (519.56, 545.95, 12) mm, rotated rx -180 ry 0 rz 160 deg; joints [11.444, 81.881, -21.738, -144.815, 64.866, 163.33]
  Set speed (17.4 mm/s)
  Call Extruder(241.03651)
  MoveL 996 to (519.07, 546.15, 12) mm, rotated rx 180 ry 0 rz 160 deg; joints [11.479, 81.804, -21.565, -144.804, 64.956, 163.375]
  Set speed (17.5 mm/s)
  Call Extruder(247.36599)
  MoveL 997 to (517.25, 546.87, 12) mm, rotated rx 180 ry 0 rz 160 deg; joints [11.607, 81.518, -20.914, -144.766, 65.289, 163.55]
  Call Extruder(253.95966)
  MoveL 998 to (515.32, 547.53, 12) mm, rotated rx 180 ry 0 rz 160 deg; joints [11.733, 81.217, -20.228, -144.735, 65.639, 163.739]
  Call Extruder(260.54470)
  MoveL 999 to (513.37, 548.12, 12) mm, rotated rx 180 ry 0 rz 160 deg; joints [11.85, 80.915, -19.537, -144.712, 65.99, 163.935]
  Set speed (17.4 mm/s)
  Call Extruder(263.42897)
  MoveL 1000 to (512.51, 548.35, 12) mm, rotated rx 180 ry 0 rz 160 deg; joints [11.899, 80.782, -19.231, -144.705, 66.144, 164.023]
  Set speed (17.4 mm/s)
  Call Extruder(267.12494)
  MoveL 1001 to (511.4, 548.62, 12) mm, rotated rx -180 ry 0 rz 160 deg; joints [11.959, 80.612, -18.84, -144.698, 66.341, 164.138]
  Set speed (17.5 mm/s)
  Call Extruder(273.88789)
  MoveL 1002 to (509.35, 549.06, 12) mm, rotated rx 180 ry 0 rz 160 deg; joints [12.063, 80.299, -18.118, -144.692, 66.703, 164.352]
  Set speed (17.5 mm/s)
  Call Extruder(280.54174)
  MoveL 1003 to (507.32, 549.4, 12) mm, rotated rx -180 ry 0 rz 160 deg; joints [12.156, 79.991, -17.404, -144.694, 67.059, 164.568]
  Set speed (17.5 mm/s)
  Call Extruder(287.07280)
  MoveL 1004 to (505.31, 549.65, 12) mm, rotated rx 180 ry 0 rz 160 deg; joints [12.239, 79.689, -16.701, -144.705, 67.408, 164.786]
  Set speed (17.5 mm/s)
  Call Extruder(293.70817)
  MoveL 1005 to (503.27, 549.83, 12) mm, rotated rx 180 ry 0 rz 160 deg; joints [12.314, 79.383, -15.986, -144.724, 67.762, 165.012]
  Set speed (17.5 mm/s)
  Call Extruder(300.36233)
  MoveL 1006 to (501.21, 549.92, 12) mm, rotated rx -180 ry 0 rz 160 deg; joints [12.38, 79.077, -15.268, -144.752, 68.115, 165.243]
  Set speed (17.5 mm/s)
  Call Extruder(306.78243)
  MoveL 1007 to (499.22, 549.93, 12) mm, rotated rx 180 ry 0 rz 160 deg; joints [12.434, 78.783, -14.577, -144.787, 68.454, 165.469]
  Set speed (10.0 mm/s)
  MoveL 1008 to (499.22, 549.93, 16) mm, rotated rx -180 ry 0 rz 160 deg; joints [12.434, 78.04, -14, -144.749, 68.317, 165.365]
  Set speed (120.0 mm/s)
  MoveL 1009 to (499.18, 550.92, 16) mm, rotated rx -180 ry 0 rz 160 deg; joints [12.556, 78.066, -14.061, -144.614, 68.32, 165.297]
  Set speed (17.5 mm/s)
  Call Extruder(313.58300)
  MoveL 1010 to (497.07, 550.85, 16) mm, rotated rx -180 ry 0 rz 160 deg; joints [12.604, 77.757, -13.333, -144.66, 68.674, 165.54]
  Set speed (17.5 mm/s)
  Call Extruder(320.32128)
  MoveL 1011 to (494.99, 550.68, 16) mm, rotated rx -180 ry 0 rz 160 deg; joints [12.641, 77.454, -12.615, -144.714, 69.022, 165.783]
  Set speed (17.5 mm/s)
  Call Extruder(326.97851)
  MoveL 1012 to (492.95, 550.44, 16) mm, rotated rx -180 ry 0 rz 160 deg; joints [12.667, 77.157, -11.909, -144.776, 69.362, 166.026]
  Set speed (17.5 mm/s)
  Call Extruder(333.68435)
  MoveL 1013 to (490.89, 550.11, 16) mm, rotated rx 180 ry 0 rz 160 deg; joints [12.684, 76.862, -11.204, -144.847, 69.702, 166.272]
  Set speed (17.5 mm/s)
  Call Extruder(340.51818)
  MoveL 1014 to (488.82, 549.69, 16) mm, rotated rx 180 ry 0 rz 160 deg; joints [12.689, 76.565, -10.49, -144.929, 70.043, 166.525]
  Set speed (17.5 mm/s)
  Call Extruder(346.95865)
  MoveL 1015 to (486.88, 549.21, 16) mm, rotated rx 180 ry 0 rz 160 deg; joints [12.684, 76.29, -9.825, -145.015, 70.362, 166.765]
  Set speed (17.5 mm/s)
  Call Extruder(350.52877)
  MoveL 1016 to (485.82, 548.91, 16) mm, rotated rx 180 ry 0 rz 160 deg; joints [12.677, 76.139, -9.459, -145.067, 70.536, 166.898]
  Set speed (17.5 mm/s)
  Call Extruder(353.73931)
  MoveL 1017 to (484.87, 548.63, 16) mm, rotated rx -180 ry 0 rz 160 deg; joints [12.668, 76.004, -9.133, -145.114, 70.691, 167.017]
  Set speed (17.5 mm/s)
  Call Extruder(360.51053)
  MoveL 1018 to (482.88, 547.97, 16) mm, rotated rx -180 ry 0 rz 160 deg; joints [12.641, 75.724, -8.45, -145.222, 71.016, 167.27]
  Set speed (17.5 mm/s)
  Call Extruder(362.35642)
  MoveL 1019 to (482.34, 547.77, 16) mm, rotated rx 180 ry 0 rz 160 deg; joints [12.632, 75.649, -8.266, -145.253, 71.103, 167.339]
  Set speed (17.5 mm/s)
  Call Extruder(367.30805)
  MoveL 1020 to (480.91, 547.22, 16) mm, rotated rx 180 ry 0 rz 160 deg; joints [12.602, 75.449, -7.775, -145.34, 71.336, 167.523]
  Set speed (17.4 mm/s)
  Call Extruder(372.34813)
  MoveL 1021 to (479.48, 546.62, 16) mm, rotated rx -180 ry 0 rz 160 deg; joints [12.566, 75.248, -7.281, -145.433, 71.569, 167.711]
  Call Extruder(377.38557)
  MoveL 1022 to (478.06, 545.97, 16) mm, rotated rx -180 ry 0 rz 160 deg; joints [12.523, 75.051, -6.795, -145.531, 71.799, 167.897]
  Set speed (17.5 mm/s)
  Call Extruder(380.80463)
  MoveL 1023 to (477.11, 545.5, 16) mm, rotated rx 180 ry 0 rz 160 deg; joints [12.49, 74.919, -6.468, -145.601, 71.953, 168.024]
  Call Extruder(384.11279)
  MoveL 1024 to (476.2, 545.03, 16) mm, rotated rx -180 ry 0 rz 160 deg; joints [12.456, 74.793, -6.154, -145.671, 72.1, 168.146]
  Set speed (17.5 mm/s)
  Call Extruder(387.48632)
  MoveL 1025 to (475.28, 544.53, 16) mm, rotated rx 180 ry 0 rz 160 deg; joints [12.418, 74.666, -5.838, -145.744, 72.249, 168.27]
  Set speed (17.5 mm/s)
  Call Extruder(390.80635)
  MoveL 1026 to (474.39, 544.02, 16) mm, rotated rx 180 ry 0 rz 160 deg; joints [12.378, 74.542, -5.529, -145.818, 72.394, 168.392]
  Set speed (17.5 mm/s)
  Call Extruder(394.19827)
  MoveL 1027 to (473.49, 543.48, 16) mm, rotated rx -180 ry 0 rz 160 deg; joints [12.334, 74.418, -5.217, -145.897, 72.54, 168.516]
  Set speed (17.5 mm/s)
  Call Extruder(397.59080)
  MoveL 1028 to (472.59, 542.93, 16) mm, rotated rx 180 ry 0 rz 160 deg; joints [12.287, 74.295, -4.909, -145.977, 72.684, 168.639]
  Set speed (17.5 mm/s)
  Call Extruder(400.94840)
  MoveL 1029 to (471.72, 542.36, 16) mm, rotated rx 180 ry 0 rz 160 deg; joints [12.238, 74.175, -4.608, -146.059, 72.825, 168.76]
  Set speed (17.5 mm/s)
  Call Extruder(404.33716)
  MoveL 1030 to (470.86, 541.77, 16) mm, rotated rx 180 ry 0 rz 160 deg; joints [12.185, 74.056, -4.307, -146.144, 72.966, 168.882]
  Set speed (17.5 mm/s)
  Call Extruder(407.70019)
  MoveL 1031 to (470.01, 541.16, 16) mm, rotated rx 180 ry 0 rz 160 deg; joints [12.13, 73.94, -4.013, -146.231, 73.103, 169.002]
  Set speed (17.5 mm/s)
  Call Extruder(411.56207)
  MoveL 1032 to (469.05, 540.45, 16) mm, rotated rx -180 ry 0 rz 160 deg; joints [12.064, 73.808, -3.68, -146.333, 73.258, 169.139]
  Set speed (17.5 mm/s)
  Call Extruder(414.44492)
  MoveL 1033 to (468.34, 539.9, 16) mm, rotated rx 180 ry 0 rz 160 deg; joints [12.011, 73.712, -3.434, -146.412, 73.372, 169.24]
  Set speed (17.5 mm/s)
  Call Extruder(417.78281)
  MoveL 1034 to (467.54, 539.25, 16) mm, rotated rx 180 ry 0 rz 160 deg; joints [11.948, 73.602, -3.155, -146.505, 73.502, 169.357]
  Set speed (17.5 mm/s)
  Call Extruder(421.08188)
  MoveL 1035 to (466.76, 538.59, 16) mm, rotated rx 180 ry 0 rz 160 deg; joints [11.883, 73.495, -2.881, -146.598, 73.629, 169.471]
  Set speed (17.5 mm/s)
  Call Extruder(424.50347)
  MoveL 1036 to (465.96, 537.89, 16) mm, rotated rx -180 ry 0 rz 160 deg; joints [11.812, 73.386, -2.603, -146.698, 73.758, 169.588]
  Set speed (17.5 mm/s)
  Call Extruder(427.79018)
  MoveL 1037 to (465.21, 537.2, 16) mm, rotated rx -180 ry 0 rz 160 deg; joints [11.742, 73.283, -2.339, -146.795, 73.88, 169.7]
  Call Extruder(431.22298)
  MoveL 1038 to (464.44, 536.47, 16) mm, rotated rx 180 ry 0 rz 160 deg; joints [11.666, 73.178, -2.068, -146.899, 74.005, 169.816]
  Set speed (17.5 mm/s)
  Call Extruder(434.57202)
  MoveL 1039 to (463.71, 535.73, 16) mm, rotated rx -180 ry 0 rz 160 deg; joints [11.589, 73.077, -1.809, -147.003, 74.124, 169.928]
  Set speed (17.5 mm/s)
  Call Extruder(438.03932)
  MoveL 1040 to (462.96, 534.96, 16) mm, rotated rx -180 ry 0 rz 160 deg; joints [11.506, 72.975, -1.545, -147.113, 74.246, 170.042]
  Set speed (17.5 mm/s)
  Call Extruder(441.29679)
  MoveL 1041 to (462.28, 534.22, 16) mm, rotated rx 180 ry 0 rz 160 deg; joints [11.426, 72.881, -1.302, -147.218, 74.357, 170.149]
  Set speed (17.5 mm/s)
  Call Extruder(446.93110)
  MoveL 1042 to (461.13, 532.91, 16) mm, rotated rx 180 ry 0 rz 160 deg; joints [11.281, 72.724, -0.892, -147.404, 74.545, 170.33]
  Set speed (17.5 mm/s)
  Call Extruder(451.31817)
  MoveL 1043 to (460.26, 531.86, 16) mm, rotated rx -180 ry 0 rz 160 deg; joints [11.163, 72.605, -0.582, -147.553, 74.687, 170.469]
  Set speed (17.5 mm/s)
  Call Extruder(454.76189)
  MoveL 1044 to (459.61, 531.02, 16) mm, rotated rx 180 ry 0 rz 160 deg; joints [11.067, 72.514, -0.345, -147.672, 74.795, 170.576]
  Set speed (17.5 mm/s)
  Call Extruder(458.13893)
  MoveL 1045 to (458.98, 530.18, 16) mm, rotated rx 180 ry 0 rz 160 deg; joints [10.97, 72.428, -0.118, -147.791, 74.898, 170.679]
  Set speed (17.5 mm/s)
  Call Extruder(461.47262)
  MoveL 1046 to (458.37, 529.35, 16) mm, rotated rx -180 ry 0 rz 160 deg; joints [10.873, 72.344, 0.102, -147.91, 74.997, 170.78]
  Call Extruder(464.83673)
  MoveL 1047 to (457.78, 528.49, 16) mm, rotated rx 180 ry 0 rz 160 deg; joints [10.772, 72.262, 0.318, -148.033, 75.095, 170.88]
  Set speed (17.5 mm/s)
  Call Extruder(468.20179)
  MoveL 1048 to (457.21, 527.62, 16) mm, rotated rx -180 ry 0 rz 160 deg; joints [10.668, 72.182, 0.529, -148.157, 75.189, 170.979]
  Set speed (17.5 mm/s)
  Call Extruder(471.65450)
  MoveL 1049 to (456.64, 526.71, 16) mm, rotated rx 180 ry 0 rz 160 deg; joints [10.56, 72.102, 0.74, -148.286, 75.284, 171.079]
  Set speed (17.5 mm/s)
  Call Extruder(474.89371)
  MoveL 1050 to (456.12, 525.85, 16) mm, rotated rx -180 ry 0 rz 160 deg; joints [10.455, 72.03, 0.932, -148.409, 75.369, 171.17]
  Set speed (17.5 mm/s)
  Call Extruder(478.28554)
  MoveL 1051 to (455.6, 524.94, 16) mm, rotated rx -180 ry 0 rz 160 deg; joints [10.344, 71.956, 1.128, -148.539, 75.457, 171.265]
  Call Extruder(481.62435)
  MoveL 1052 to (455.1, 524.04, 16) mm, rotated rx 180 ry 0 rz 160 deg; joints [10.232, 71.886, 1.315, -148.669, 75.539, 171.356]
  Call Extruder(484.99783)
  MoveL 1053 to (454.62, 523.11, 16) mm, rotated rx 180 ry 0 rz 160 deg; joints [10.117, 71.817, 1.499, -148.802, 75.62, 171.447]
  Set speed (17.5 mm/s)
  Call Extruder(488.42921)
  MoveL 1054 to (454.14, 522.16, 16) mm, rotated rx -180 ry 0 rz 160 deg; joints [9.997, 71.749, 1.679, -148.939, 75.699, 171.538]
  Call Extruder(495.10061)
  MoveL 1055 to (453.28, 520.28, 16) mm, rotated rx -180 ry 0 rz 160 deg; joints [9.759, 71.624, 2.014, -149.21, 75.845, 171.709]
  Set speed (17.5 mm/s)
  Call Extruder(498.56852)
  MoveL 1056 to (452.87, 519.29, 16) mm, rotated rx -180 ry 0 rz 160 deg; joints [9.632, 71.563, 2.177, -149.353, 75.914, 171.795]
  Set speed (17.4 mm/s)
  Call Extruder(503.66353)
  MoveL 1057 to (452.29, 517.83, 16) mm, rotated rx -180 ry 0 rz 160 deg; joints [9.442, 71.478, 2.407, -149.565, 76.012, 171.917]
  Set speed (17.4 mm/s)
  Call Extruder(508.79051)
  MoveL 1058 to (451.76, 516.33, 16) mm, rotated rx 180 ry 0 rz 160 deg; joints [9.247, 71.397, 2.625, -149.781, 76.103, 172.036]
  Set speed (17.5 mm/s)
  Call Extruder(515.41803)
  MoveL 1059 to (451.14, 514.38, 16) mm, rotated rx 180 ry 0 rz 160 deg; joints [8.988, 71.301, 2.885, -150.065, 76.209, 172.184]
  Call Extruder(521.98039)
  MoveL 1060 to (450.61, 512.42, 16) mm, rotated rx -180 ry 0 rz 160 deg; joints [8.726, 71.215, 3.118, -150.351, 76.302, 172.323]
  Set speed (17.5 mm/s)
  Call Extruder(525.48408)
  MoveL 1061 to (450.36, 511.36, 16) mm, rotated rx 180 ry 0 rz 160 deg; joints [8.583, 71.173, 3.232, -150.505, 76.345, 172.394]
  Set speed (17.5 mm/s)
  Call Extruder(528.68540)
  MoveL 1062 to (450.14, 510.4, 16) mm, rotated rx 180 ry 0 rz 160 deg; joints [8.452, 71.137, 3.331, -150.646, 76.383, 172.457]
  Set speed (17.5 mm/s)
  Call Extruder(535.63344)
  MoveL 1063 to (449.75, 508.28, 16) mm, rotated rx -180 ry 0 rz 160 deg; joints [8.163, 71.065, 3.527, -150.956, 76.453, 172.589]
  Set speed (17.5 mm/s)
  Call Extruder(542.34708)
  MoveL 1064 to (449.45, 506.22, 16) mm, rotated rx 180 ry 0 rz 160 deg; joints [7.879, 71.006, 3.689, -151.258, 76.507, 172.708]
  Set speed (17.5 mm/s)
  Call Extruder(549.08310)
  MoveL 1065 to (449.24, 504.15, 16) mm, rotated rx 180 ry 0 rz 160 deg; joints [7.59, 70.956, 3.826, -151.562, 76.547, 172.819]
  Call Extruder(555.62489)
  MoveL 1066 to (449.11, 502.12, 16) mm, rotated rx -180 ry 0 rz 160 deg; joints [7.306, 70.916, 3.934, -151.859, 76.572, 172.92]
  Set speed (17.5 mm/s)
  Call Extruder(562.43855)
  MoveL 1067 to (449.07, 500.01, 16) mm, rotated rx 180 ry 0 rz 160 deg; joints [7.008, 70.885, 4.019, -152.169, 76.583, 173.016]
  Set speed (17.5 mm/s)
  Call Extruder(568.56607)
  MoveL 1068 to (449.1, 498.12, 16) mm, rotated rx -180 ry 0 rz 160 deg; joints [6.739, 70.866, 4.073, -152.448, 76.581, 173.096]
  Set speed (17.5 mm/s)
  Call Extruder(574.54826)
  MoveL 1069 to (449.21, 496.27, 16) mm, rotated rx 180 ry 0 rz 160 deg; joints [6.474, 70.855, 4.103, -152.72, 76.566, 173.168]
  Call Extruder(580.52338)
  MoveL 1070 to (449.38, 494.42, 16) mm, rotated rx -180 ry 0 rz 160 deg; joints [6.21, 70.851, 4.113, -152.991, 76.541, 173.234]
  Call Extruder(586.64948)
  MoveL 1071 to (449.62, 492.54, 16) mm, rotated rx -180 ry 0 rz 160 deg; joints [5.939, 70.855, 4.101, -153.267, 76.502, 173.295]
  Set speed (17.5 mm/s)
  Call Extruder(592.79375)
  MoveL 1072 to (449.93, 490.66, 16) mm, rotated rx 180 ry 0 rz 160 deg; joints [5.668, 70.867, 4.068, -153.541, 76.452, 173.35]
  Set speed (17.5 mm/s)
  Call Extruder(598.71057)
  MoveL 1073 to (450.3, 488.87, 16) mm, rotated rx 180 ry 0 rz 160 deg; joints [5.408, 70.887, 4.013, -153.803, 76.391, 173.397]
  Set speed (17.5 mm/s)
  Call Extruder(604.81441)
  MoveL 1074 to (450.75, 487.03, 16) mm, rotated rx -180 ry 0 rz 160 deg; joints [5.141, 70.915, 3.936, -154.071, 76.316, 173.439]
  Set speed (17.5 mm/s)
  Call Extruder(610.86663)
  MoveL 1075 to (451.26, 485.23, 16) mm, rotated rx 180 ry 0 rz 160 deg; joints [4.878, 70.951, 3.839, -154.333, 76.23, 173.475]
  Set speed (17.5 mm/s)
  Call Extruder(616.73710)
  MoveL 1076 to (451.82, 483.5, 16) mm, rotated rx -180 ry 0 rz 160 deg; joints [4.626, 70.993, 3.723, -154.583, 76.136, 173.504]
  Set speed (17.5 mm/s)
  Call Extruder(622.96146)
  MoveL 1077 to (452.48, 481.68, 16) mm, rotated rx -180 ry 0 rz 160 deg; joints [4.361, 71.046, 3.579, -154.845, 76.023, 173.529]
  Set speed (17.5 mm/s)
  Call Extruder(629.10427)
  MoveL 1078 to (453.2, 479.92, 16) mm, rotated rx -180 ry 0 rz 160 deg; joints [4.104, 71.106, 3.415, -155.097, 75.9, 173.548]
  Call Extruder(635.10844)
  MoveL 1079 to (453.96, 478.23, 16) mm, rotated rx -180 ry 0 rz 160 deg; joints [3.857, 71.172, 3.235, -155.339, 75.769, 173.56]
  Set speed (17.5 mm/s)
  Call Extruder(641.16131)
  MoveL 1080 to (454.79, 476.55, 16) mm, rotated rx 180 ry 0 rz 160 deg; joints [3.611, 71.247, 3.032, -155.576, 75.625, 173.567]
  Call Extruder(647.10344)
  MoveL 1081 to (455.67, 474.93, 16) mm, rotated rx -180 ry 0 rz 160 deg; joints [3.376, 71.328, 2.813, -155.804, 75.472, 173.569]
  Call Extruder(653.06625)
  MoveL 1082 to (456.61, 473.34, 16) mm, rotated rx 180 ry 0 rz 160 deg; joints [3.144, 71.416, 2.574, -156.026, 75.309, 173.566]
  Call Extruder(659.45229)
  MoveL 1083 to (457.67, 471.67, 16) mm, rotated rx -180 ry 0 rz 160 deg; joints [2.902, 71.519, 2.297, -156.256, 75.122, 173.556]
  Set speed (17.5 mm/s)
  Call Extruder(665.32584)
  MoveL 1084 to (458.71, 470.18, 16) mm, rotated rx 180 ry 0 rz 160 deg; joints [2.685, 71.621, 2.022, -156.46, 74.94, 173.542]
  Set speed (17.5 mm/s)
  Call Extruder(671.46768)
  MoveL 1085 to (459.86, 468.66, 16) mm, rotated rx -180 ry 0 rz 160 deg; joints [2.465, 71.735, 1.716, -156.666, 74.739, 173.522]
  Set speed (17.5 mm/s)
  Call Extruder(678.46535)
  MoveL 1086 to (461.22, 466.97, 16) mm, rotated rx -180 ry 0 rz 160 deg; joints [2.222, 71.875, 1.344, -156.891, 74.498, 173.494]
  Call Extruder(679.84425)
  MoveL 1087 to (461.51, 466.66, 16) mm, rotated rx -180 ry 0 rz 160 deg; joints [2.177, 71.905, 1.265, -156.933, 74.447, 173.486]
  Set speed (17.5 mm/s)
  Call Extruder(683.40151)
  MoveL 1088 to (462.24, 465.83, 16) mm, rotated rx 180 ry 0 rz 160 deg; joints [2.058, 71.98, 1.065, -157.042, 74.319, 173.468]
  Call Extruder(689.62345)
  MoveL 1089 to (463.56, 464.42, 16) mm, rotated rx 180 ry 0 rz 160 deg; joints [1.856, 72.118, 0.699, -157.225, 74.086, 173.433]
  Call Extruder(695.50895)
  MoveL 1090 to (464.85, 463.14, 16) mm, rotated rx 180 ry 0 rz 160 deg; joints [1.674, 72.256, 0.334, -157.388, 73.856, 173.394]
  Call Extruder(701.58704)
  MoveL 1091 to (466.24, 461.87, 16) mm, rotated rx -180 ry 0 rz 160 deg; joints [1.493, 72.406, -0.06, -157.548, 73.609, 173.349]
  Set speed (17.5 mm/s)
  Call Extruder(707.79963)
  MoveL 1092 to (467.7, 460.62, 16) mm, rotated rx 180 ry 0 rz 160 deg; joints [1.316, 72.566, -0.479, -157.702, 73.349, 173.298]
  Set speed (17.5 mm/s)
  Call Extruder(714.13257)
  MoveL 1093 to (469.24, 459.41, 16) mm, rotated rx 180 ry 0 rz 160 deg; joints [1.145, 72.736, -0.925, -157.848, 73.075, 173.241]
  Call Extruder(719.86338)
  MoveL 1094 to (470.68, 458.36, 16) mm, rotated rx -180 ry 0 rz 160 deg; joints [0.998, 72.897, -1.343, -157.971, 72.819, 173.184]
  Set speed (17.5 mm/s)
  Call Extruder(725.78899)
  MoveL 1095 to (472.19, 457.33, 16) mm, rotated rx 180 ry 0 rz 160 deg; joints [0.855, 73.07, -1.791, -158.088, 72.547, 173.121]
  Set speed (17.5 mm/s)
  Call Extruder(732.01007)
  MoveL 1096 to (473.83, 456.31, 16) mm, rotated rx 180 ry 0 rz 160 deg; joints [0.713, 73.259, -2.276, -158.201, 72.255, 173.05]
  Set speed (17.5 mm/s)
  Call Extruder(738.06083)
  MoveL 1097 to (475.45, 455.38, 16) mm, rotated rx -180 ry 0 rz 160 deg; joints [0.585, 73.448, -2.762, -158.299, 71.963, 172.975]
  Set speed (17.5 mm/s)
  Call Extruder(744.97750)
  MoveL 1098 to (477.35, 454.38, 16) mm, rotated rx 180 ry 0 rz 160 deg; joints [0.448, 73.672, -3.334, -158.399, 71.623, 172.885]
  Set speed (17.5 mm/s)
  Call Extruder(750.17427)
  MoveL 1099 to (478.8, 453.69, 16) mm, rotated rx -180 ry 0 rz 160 deg; joints [0.355, 73.846, -3.776, -158.464, 71.362, 172.812]
  Set speed (17.5 mm/s)
  Call Extruder(756.21836)
  MoveL 1100 to (480.52, 452.95, 16) mm, rotated rx 180 ry 0 rz 160 deg; joints [0.254, 74.054, -4.302, -158.53, 71.053, 172.723]
  Call Extruder(762.20586)
  MoveL 1101 to (482.24, 452.26, 16) mm, rotated rx 180 ry 0 rz 160 deg; joints [0.162, 74.265, -4.835, -158.586, 70.742, 172.63]
  Set speed (17.5 mm/s)
  Call Extruder(768.32214)
  MoveL 1102 to (484.03, 451.64, 16) mm, rotated rx 180 ry 0 rz 160 deg; joints [0.079, 74.487, -5.392, -158.63, 70.42, 172.53]
  Set speed (17.5 mm/s)
  Call Extruder(774.30251)
  MoveL 1103 to (485.8, 451.09, 16) mm, rotated rx -180 ry 0 rz 160 deg; joints [0.006, 74.71, -5.946, -158.663, 70.101, 172.427]
  Set speed (17.5 mm/s)
  Call Extruder(780.34628)
  MoveL 1104 to (487.61, 450.6, 16) mm, rotated rx -180 ry 0 rz 160 deg; joints [-0.058, 74.939, -6.518, -158.686, 69.774, 172.318]
  Set speed (17.5 mm/s)
  Call Extruder(786.49451)
  MoveL 1105 to (489.46, 450.17, 16) mm, rotated rx 180 ry 0 rz 160 deg; joints [-0.113, 75.179, -7.11, -158.697, 69.438, 172.201]
  Call Extruder(792.46948)
  MoveL 1106 to (491.28, 449.82, 16) mm, rotated rx -180 ry 0 rz 160 deg; joints [-0.159, 75.416, -7.694, -158.697, 69.109, 172.084]
  Set speed (17.5 mm/s)
  Call Extruder(798.18195)
  MoveL 1107 to (493.03, 449.55, 16) mm, rotated rx 180 ry 0 rz 160 deg; joints [-0.193, 75.647, -8.26, -158.687, 68.791, 171.966]
  Set speed (17.5 mm/s)
  Call Extruder(804.61428)
  MoveL 1108 to (495.01, 449.32, 16) mm, rotated rx 180 ry 0 rz 160 deg; joints [-0.223, 75.911, -8.906, -158.664, 68.432, 171.829]
  Set speed (17.5 mm/s)
  Call Extruder(810.61991)
  MoveL 1109 to (496.86, 449.17, 16) mm, rotated rx 180 ry 0 rz 160 deg; joints [-0.241, 76.162, -9.517, -158.631, 68.095, 171.695]
  Set speed (17.5 mm/s)
  Call Extruder(816.77165)
  MoveL 1110 to (498.76, 449.09, 16) mm, rotated rx -180 ry 0 rz 160 deg; joints [-0.25, 76.424, -10.149, -158.586, 67.748, 171.553]
  Set speed (17.5 mm/s)
  Call Extruder(822.74867)
  MoveL 1111 to (500.62, 449.07, 16) mm, rotated rx 180 ry 0 rz 160 deg; joints [-0.251, 76.682, -10.77, -158.532, 67.41, 171.409]
  Set speed (17.5 mm/s)
  Call Extruder(828.68751)
  MoveL 1112 to (502.46, 449.13, 16) mm, rotated rx -180 ry 0 rz 160 deg; joints [-0.243, 76.941, -11.392, -158.467, 67.074, 171.262]
  Set speed (17.5 mm/s)
  Call Extruder(834.85210)
  MoveL 1113 to (504.36, 449.26, 16) mm, rotated rx -180 ry 0 rz 160 deg; joints [-0.226, 77.213, -12.042, -158.39, 66.725, 171.104]
  Set speed (17.5 mm/s)
  Call Extruder(840.96812)
  MoveL 1114 to (506.25, 449.45, 16) mm, rotated rx 180 ry 0 rz 160 deg; joints [-0.2, 77.486, -12.691, -158.302, 66.379, 170.941]
  Set speed (17.5 mm/s)
  Call Extruder(846.86486)
  MoveL 1115 to (508.06, 449.71, 16) mm, rotated rx -180 ry 0 rz 160 deg; joints [-0.167, 77.752, -13.32, -158.207, 66.047, 170.78]
  Set speed (17.5 mm/s)
  Call Extruder(853.07190)
  MoveL 1116 to (509.95, 450.05, 16) mm, rotated rx -180 ry 0 rz 160 deg; joints [-0.124, 78.033, -13.984, -158.097, 65.699, 170.605]
  Call Extruder(858.91147)
  MoveL 1117 to (511.72, 450.44, 16) mm, rotated rx 180 ry 0 rz 160 deg; joints [-0.075, 78.3, -14.611, -157.983, 65.373, 170.435]
  Set speed (17.5 mm/s)
  Call Extruder(865.02699)
  MoveL 1118 to (513.55, 450.91, 16) mm, rotated rx 180 ry 0 rz 160 deg; joints [-0.017, 78.581, -15.268, -157.854, 65.034, 170.253]
  Call Extruder(871.15278)
  MoveL 1119 to (515.37, 451.45, 16) mm, rotated rx -180 ry 0 rz 160 deg; joints [0.05, 78.863, -15.926, -157.715, 64.697, 170.065]
  Set speed (17.5 mm/s)
  Call Extruder(877.28716)
  MoveL 1120 to (517.17, 452.05, 16) mm, rotated rx -180 ry 0 rz 160 deg; joints [0.124, 79.147, -16.585, -157.566, 64.363, 169.872]
  Set speed (17.5 mm/s)
  Call Extruder(883.24316)
  MoveL 1121 to (518.9, 452.71, 16) mm, rotated rx -180 ry 0 rz 160 deg; joints [0.204, 79.423, -17.223, -157.412, 64.043, 169.68]
  Set speed (17.5 mm/s)
  Call Extruder(889.38332)
  MoveL 1122 to (520.65, 453.45, 16) mm, rotated rx 180 ry 0 rz 160 deg; joints [0.293, 79.707, -17.878, -157.244, 63.717, 169.478]
  Set speed (17.5 mm/s)
  Call Extruder(895.43566)
  MoveL 1123 to (522.35, 454.24, 16) mm, rotated rx 180 ry 0 rz 160 deg; joints [0.388, 79.987, -18.52, -157.07, 63.401, 169.274]
  Call Extruder(901.36027)
  MoveL 1124 to (523.99, 455.07, 16) mm, rotated rx 180 ry 0 rz 160 deg; joints [0.488, 80.26, -19.145, -156.89, 63.096, 169.071]
  Set speed (17.5 mm/s)
  Call Extruder(907.54881)
  MoveL 1125 to (525.66, 456.01, 16) mm, rotated rx -180 ry 0 rz 160 deg; joints [0.599, 80.544, -19.793, -156.695, 62.782, 168.854]
  Call Extruder(913.49773)
  MoveL 1126 to (527.23, 456.96, 16) mm, rotated rx -180 ry 0 rz 160 deg; joints [0.712, 80.815, -20.41, -156.499, 62.488, 168.642]
  Set speed (17.5 mm/s)
  Call Extruder(919.64017)
  MoveL 1127 to (528.82, 458.01, 16) mm, rotated rx -180 ry 0 rz 160 deg; joints [0.835, 81.093, -21.04, -156.289, 62.189, 168.42]
  Set speed (17.5 mm/s)
  Call Extruder(925.59884)
  MoveL 1128 to (530.33, 459.08, 16) mm, rotated rx -180 ry 0 rz 160 deg; joints [0.96, 81.36, -21.643, -156.078, 61.907, 168.201]
  Set speed (17.5 mm/s)
  Call Extruder(931.65208)
  MoveL 1129 to (531.81, 460.23, 16) mm, rotated rx 180 ry 0 rz 160 deg; joints [1.094, 81.629, -22.248, -155.856, 61.628, 167.975]
  Set speed (17.5 mm/s)
  Call Extruder(937.75693)
  MoveL 1130 to (533.27, 461.44, 16) mm, rotated rx 180 ry 0 rz 160 deg; joints [1.234, 81.897, -22.849, -155.626, 61.354, 167.745]
  Set speed (17.5 mm/s)
  Call Extruder(943.68461)
  MoveL 1131 to (534.64, 462.66, 16) mm, rotated rx 180 ry 0 rz 160 deg; joints [1.375, 82.152, -23.421, -155.396, 61.096, 167.52]
  Set speed (17.5 mm/s)
  Call Extruder(949.87674)
  MoveL 1132 to (536.02, 463.99, 16) mm, rotated rx 180 ry 0 rz 160 deg; joints [1.529, 82.415, -24.007, -155.15, 60.835, 167.282]
  Call Extruder(953.15618)
  MoveL 1133 to (536.73, 464.72, 16) mm, rotated rx -180 ry 0 rz 160 deg; joints [1.612, 82.552, -24.312, -155.017, 60.701, 167.155]
  Set speed (17.5 mm/s)
  Call Extruder(956.44654)
  MoveL 1134 to (537.43, 465.46, 16) mm, rotated rx 180 ry 0 rz 160 deg; joints [1.697, 82.688, -24.615, -154.883, 60.569, 167.028]
  Set speed (17.5 mm/s)
  Call Extruder(959.83210)
  MoveL 1135 to (538.13, 466.24, 16) mm, rotated rx -180 ry 0 rz 160 deg; joints [1.786, 82.826, -24.921, -154.743, 60.437, 166.897]
  Call Extruder(963.19392)
  MoveL 1136 to (538.81, 467.03, 16) mm, rotated rx 180 ry 0 rz 160 deg; joints [1.876, 82.962, -25.222, -154.602, 60.308, 166.766]
  Set speed (17.5 mm/s)
  Call Extruder(966.60977)
  MoveL 1137 to (539.49, 467.84, 16) mm, rotated rx 180 ry 0 rz 160 deg; joints [1.968, 83.097, -25.521, -154.457, 60.181, 166.633]
  Set speed (17.5 mm/s)
  Call Extruder(969.93627)
  MoveL 1138 to (540.13, 468.64, 16) mm, rotated rx -180 ry 0 rz 160 deg; joints [2.06, 83.228, -25.81, -154.316, 60.06, 166.503]
  Set speed (17.5 mm/s)
  Call Extruder(973.31274)
  MoveL 1139 to (540.77, 469.48, 16) mm, rotated rx 180 ry 0 rz 160 deg; joints [2.154, 83.357, -26.097, -154.17, 59.941, 166.371]
  Set speed (17.5 mm/s)
  Call Extruder(976.62924)
  MoveL 1140 to (541.38, 470.31, 16) mm, rotated rx -180 ry 0 rz 160 deg; joints [2.248, 83.483, -26.374, -154.026, 59.827, 166.241]
  Set speed (17.5 mm/s)
  Call Extruder(980.01829)
  MoveL 1141 to (541.98, 471.16, 16) mm, rotated rx 180 ry 0 rz 160 deg; joints [2.345, 83.609, -26.652, -153.878, 59.714, 166.109]
  Set speed (17.5 mm/s)
  Call Extruder(983.45435)
  MoveL 1142 to (542.58, 472.05, 16) mm, rotated rx -180 ry 0 rz 160 deg; joints [2.445, 83.735, -26.93, -153.727, 59.602, 165.975]
  Set speed (17.5 mm/s)
  Call Extruder(986.76532)
  MoveL 1143 to (543.13, 472.91, 16) mm, rotated rx 180 ry 0 rz 160 deg; joints [2.543, 83.853, -27.189, -153.58, 59.499, 165.847]
  Set speed (17.5 mm/s)
  Call Extruder(990.13044)
  MoveL 1144 to (543.67, 473.8, 16) mm, rotated rx 180 ry 0 rz 160 deg; joints [2.643, 83.971, -27.448, -153.43, 59.397, 165.717]
  Set speed (17.5 mm/s)
  Call Extruder(993.46029)
  MoveL 1145 to (544.19, 474.69, 16) mm, rotated rx -180 ry 0 rz 160 deg; joints [2.743, 84.086, -27.699, -153.281, 59.3, 165.588]
  Set speed (17.5 mm/s)
  Call Extruder(998.85620)
  MoveL 1146 to (545, 476.15, 16) mm, rotated rx -180 ry 0 rz 160 deg; joints [2.908, 84.266, -28.093, -153.038, 59.15, 165.38]
  Set speed (17.5 mm/s)
  Call Extruder(1003.57253)
  MoveL 1147 to (545.66, 477.45, 16) mm, rotated rx -180 ry 0 rz 160 deg; joints [3.054, 84.416, -28.422, -152.825, 59.029, 165.201]
  Set speed (17.5 mm/s)
  Call Extruder(1006.90451)
  MoveL 1148 to (546.11, 478.38, 16) mm, rotated rx 180 ry 0 rz 160 deg; joints [3.158, 84.52, -28.647, -152.673, 58.947, 165.075]
  Set speed (17.5 mm/s)
  Call Extruder(1010.34170)
  MoveL 1149 to (546.55, 479.35, 16) mm, rotated rx 180 ry 0 rz 160 deg; joints [3.267, 84.623, -28.873, -152.517, 58.866, 164.946]
  Set speed (17.5 mm/s)
  Call Extruder(1013.73787)
  MoveL 1150 to (546.97, 480.31, 16) mm, rotated rx 180 ry 0 rz 160 deg; joints [3.376, 84.721, -29.087, -152.362, 58.792, 164.82]
  Set speed (17.5 mm/s)
  Call Extruder(1016.91797)
  MoveL 1151 to (547.34, 481.22, 16) mm, rotated rx -180 ry 0 rz 160 deg; joints [3.478, 84.812, -29.284, -152.217, 58.725, 164.702]
  Set speed (17.5 mm/s)
  Call Extruder(1020.46764)
  MoveL 1152 to (547.73, 482.25, 16) mm, rotated rx 180 ry 0 rz 160 deg; joints [3.593, 84.908, -29.493, -152.055, 58.655, 164.573]
  Call Extruder(1023.68738)
  MoveL 1153 to (548.07, 483.19, 16) mm, rotated rx -180 ry 0 rz 160 deg; joints [3.698, 84.994, -29.68, -151.907, 58.594, 164.456]
  Set speed (17.5 mm/s)
  Call Extruder(1027.20899)
  MoveL 1154 to (548.42, 484.22, 16) mm, rotated rx 180 ry 0 rz 160 deg; joints [3.814, 85.082, -29.871, -151.747, 58.534, 164.331]
  Set speed (17.4 mm/s)
  Call Extruder(1030.48977)
  MoveL 1155 to (548.73, 485.18, 16) mm, rotated rx -180 ry 0 rz 160 deg; joints [3.922, 85.162, -30.046, -151.597, 58.481, 164.214]
  Set speed (17.5 mm/s)
  Call Extruder(1037.31304)
  MoveL 1156 to (549.3, 487.22, 16) mm, rotated rx -180 ry 0 rz 160 deg; joints [4.15, 85.317, -30.381, -151.287, 58.385, 163.978]
  Set speed (17.5 mm/s)
  Call Extruder(1043.94080)
  MoveL 1157 to (549.77, 489.21, 16) mm, rotated rx -180 ry 0 rz 160 deg; joints [4.374, 85.453, -30.675, -150.987, 58.309, 163.756]
  Call Extruder(1050.72404)
  MoveL 1158 to (550.17, 491.28, 16) mm, rotated rx -180 ry 0 rz 160 deg; joints [4.605, 85.576, -30.942, -150.683, 58.249, 163.537]
  Set speed (17.5 mm/s)
  Call Extruder(1057.45627)
  MoveL 1159 to (550.49, 493.34, 16) mm, rotated rx -180 ry 0 rz 160 deg; joints [4.837, 85.684, -31.174, -150.383, 58.206, 163.327]
  Set speed (17.5 mm/s)
  Call Extruder(1064.28473)
  MoveL 1160 to (550.73, 495.44, 16) mm, rotated rx -180 ry 0 rz 160 deg; joints [5.074, 85.776, -31.373, -150.084, 58.182, 163.124]
  Set speed (17.5 mm/s)
  Call Extruder(1070.91155)
  MoveL 1161 to (550.87, 497.49, 16) mm, rotated rx -180 ry 0 rz 160 deg; joints [5.305, 85.849, -31.53, -149.797, 58.176, 162.937]
  Set speed (17.5 mm/s)
  Call Extruder(1077.63419)
  MoveL 1162 to (550.93, 499.57, 16) mm, rotated rx -180 ry 0 rz 160 deg; joints [5.541, 85.907, -31.654, -149.511, 58.188, 162.758]
  Set speed (17.5 mm/s)
  Call Extruder(1084.44688)
  MoveL 1163 to (550.9, 501.68, 16) mm, rotated rx 180 ry 0 rz 160 deg; joints [5.781, 85.948, -31.743, -149.227, 58.219, 162.587]
  Set speed (17.5 mm/s)
  Call Extruder(1091.08003)
  MoveL 1164 to (550.79, 503.73, 16) mm, rotated rx 180 ry 0 rz 160 deg; joints [6.015, 85.97, -31.792, -148.956, 58.267, 162.433]
  Call Extruder(1097.71652)
  MoveL 1165 to (550.6, 505.78, 16) mm, rotated rx 180 ry 0 rz 160 deg; joints [6.249, 85.977, -31.805, -148.692, 58.332, 162.291]
  Set speed (17.5 mm/s)
  Call Extruder(1104.63353)
  MoveL 1166 to (550.31, 507.9, 16) mm, rotated rx -180 ry 0 rz 160 deg; joints [6.493, 85.965, -31.781, -148.423, 58.417, 162.156]
  Set speed (17.5 mm/s)
  Call Extruder(1111.25604)
  MoveL 1167 to (549.95, 509.92, 16) mm, rotated rx -180 ry 0 rz 160 deg; joints [6.726, 85.938, -31.721, -148.173, 58.516, 162.039]
  Set speed (17.5 mm/s)
  Call Extruder(1118.03663)
  MoveL 1168 to (549.5, 511.97, 16) mm, rotated rx 180 ry 0 rz 160 deg; joints [6.965, 85.892, -31.622, -147.924, 58.635, 161.934]
  Set speed (17.5 mm/s)
  Call Extruder(1121.37330)
